Yaskawa INFORM job: DEMO_ROOF_SIDE_0625_3PAINT_37.JBI

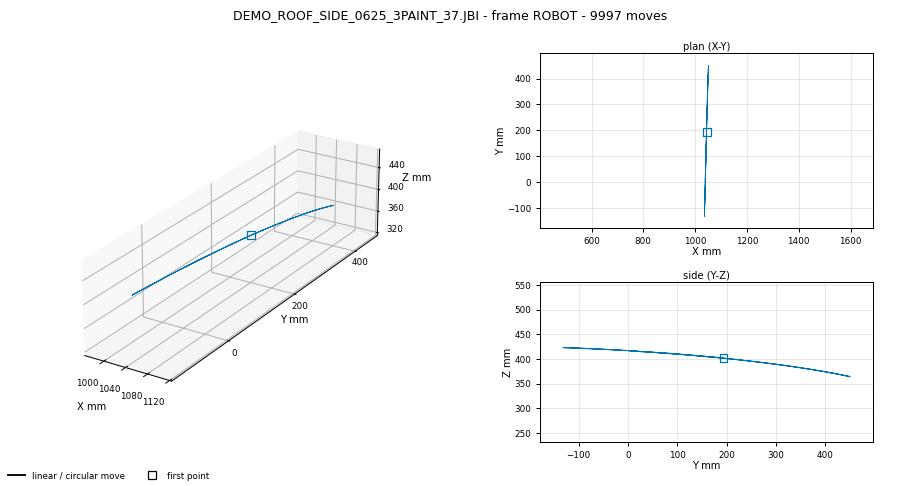
[picture p0: tool path of DEMO_ROOF_SIDE_0625_3PAINT_37.JBI in frame ROBOT, 9997 of 9997 moves have a stored position in this frame; points joined in program order, loops and branches not executed]
/JOB
//NAME DEMO_ROOF_SIDE_0625_3PAINT37
//POS
///NPOS 9997,0,0,0,0,0
///TOOL 0
///USER 0
///POSTYPE ROBOT
///RECTAN
///RCONF 1,0,0,0,0,0,0,0,0,0,0,0,0,0,0,0,0,0,0,0,0,0,0,0
C00000=1044.658,193.704,402.570,170.909,38.370,157.244
C00001=1044.653,193.455,402.594,170.907,38.368,157.244
C00002=1044.647,193.206,402.619,170.903,38.367,157.243
C00003=1044.641,192.958,402.643,170.901,38.365,157.243
C00004=1044.635,192.709,402.668,170.899,38.364,157.243
C00005=1044.628,192.460,402.692,170.895,38.362,157.242
C00006=1044.623,192.211,402.716,170.893,38.360,157.242
C00007=1044.616,191.962,402.740,170.891,38.359,157.241
C00008=1044.611,191.714,402.765,170.888,38.357,157.241
C00009=1044.604,191.465,402.789,170.885,38.355,157.241
C00010=1044.598,191.216,402.814,170.883,38.353,157.240
C00011=1044.592,190.968,402.838,170.880,38.352,157.240
C00012=1044.586,190.719,402.862,170.877,38.350,157.239
C00013=1044.580,190.470,402.886,170.875,38.348,157.239
C00014=1044.574,190.221,402.911,170.872,38.347,157.239
C00015=1044.567,189.937,402.939,170.869,38.345,157.238
C00016=1044.561,189.653,402.966,170.867,38.342,157.238
C00017=1044.553,189.368,402.994,170.863,38.341,157.237
C00018=1044.547,189.083,403.022,170.860,38.339,157.237
C00019=1044.541,188.835,403.045,170.858,38.337,157.236
C00020=1044.535,188.586,403.070,170.855,38.336,157.236
C00021=1044.529,188.337,403.094,170.853,38.334,157.236
C00022=1044.523,188.088,403.118,170.850,38.332,157.235
C00023=1044.517,187.840,403.142,170.847,38.330,157.235
C00024=1044.511,187.591,403.167,170.845,38.329,157.234
C00025=1044.505,187.343,403.191,170.843,38.327,157.234
C00026=1044.499,187.094,403.216,170.840,38.325,157.234
C00027=1044.493,186.845,403.239,170.837,38.323,157.233
C00028=1044.487,186.596,403.264,170.835,38.322,157.233
C00029=1044.481,186.347,403.287,170.832,38.320,157.232
C00030=1044.475,186.098,403.311,170.830,38.319,157.232
C00031=1044.469,185.850,403.335,170.827,38.317,157.232
C00032=1044.463,185.600,403.360,170.824,38.315,157.231
C00033=1044.457,185.352,403.383,170.822,38.313,157.231
C00034=1044.451,185.104,403.407,170.820,38.312,157.230
C00035=1044.445,184.854,403.432,170.817,38.310,157.230
C00036=1044.439,184.606,403.455,170.814,38.308,157.230
C00037=1044.433,184.357,403.480,170.812,38.307,157.229
C00038=1044.427,184.109,403.504,170.809,38.305,157.229
C00039=1044.422,183.859,403.528,170.807,38.304,157.229
C00040=1044.416,183.610,403.551,170.805,38.302,157.228
C00041=1044.409,183.361,403.575,170.801,38.300,157.228
C00042=1044.403,183.113,403.599,170.799,38.299,157.227
C00043=1044.396,182.864,403.623,170.797,38.297,157.227
C00044=1044.391,182.615,403.646,170.795,38.296,157.227
C00045=1044.384,182.366,403.670,170.791,38.294,157.226
C00046=1044.378,182.118,403.693,170.789,38.293,157.226
C00047=1044.372,181.868,403.717,170.787,38.291,157.226
C00048=1044.366,181.620,403.740,170.784,38.290,157.225
C00049=1044.358,181.371,403.764,170.781,38.289,157.225
C00050=1044.353,181.123,403.787,170.779,38.287,157.225
C00051=1044.346,180.874,403.811,170.777,38.286,157.224
C00052=1044.340,180.625,403.834,170.774,38.284,157.224
C00053=1044.334,180.376,403.857,170.771,38.283,157.224
C00054=1044.328,180.127,403.882,170.769,38.281,157.223
C00055=1044.322,179.879,403.904,170.766,38.279,157.223
C00056=1044.315,179.630,403.928,170.764,38.278,157.223
C00057=1044.309,179.381,403.951,170.762,38.276,157.222
C00058=1044.303,179.132,403.975,170.758,38.275,157.222
C00059=1044.297,178.883,403.999,170.756,38.274,157.222
C00060=1044.291,178.635,404.022,170.754,38.272,157.221
C00061=1044.284,178.386,404.045,170.752,38.271,157.221
C00062=1044.278,178.137,404.068,170.749,38.270,157.221
C00063=1044.271,177.888,404.092,170.746,38.268,157.220
C00064=1044.266,177.639,404.115,170.744,38.266,157.220
C00065=1044.260,177.391,404.139,170.741,38.265,157.219
C00066=1044.253,177.141,404.162,170.739,38.263,157.219
C00067=1044.247,176.893,404.186,170.737,38.262,157.219
C00068=1044.241,176.643,404.209,170.734,38.260,157.218
C00069=1044.235,176.394,404.232,170.731,38.259,157.218
C00070=1044.229,176.146,404.256,170.729,38.257,157.218
C00071=1044.222,175.897,404.279,170.727,38.256,157.217
C00072=1044.216,175.649,404.302,170.724,38.255,157.217
C00073=1044.210,175.400,404.325,170.722,38.253,157.217
C00074=1044.204,175.151,404.349,170.719,38.252,157.216
C00075=1044.198,174.902,404.372,170.717,38.251,157.216
C00076=1044.192,174.653,404.395,170.714,38.249,157.216
C00077=1044.186,174.405,404.419,170.712,38.248,157.215
C00078=1044.180,174.155,404.442,170.710,38.246,157.215
C00079=1044.173,173.871,404.469,170.706,38.244,157.215
C00080=1044.166,173.586,404.495,170.704,38.242,157.214
C00081=1044.158,173.301,404.521,170.701,38.241,157.214
C00082=1044.152,173.016,404.548,170.699,38.239,157.214
C00083=1044.146,172.767,404.572,170.696,38.238,157.213
C00084=1044.140,172.518,404.595,170.694,38.237,157.213
C00085=1044.133,172.270,404.618,170.692,38.235,157.212
C00086=1044.127,172.020,404.641,170.689,38.234,157.212
C00087=1044.121,171.771,404.664,170.686,38.232,157.212
C00088=1044.115,171.523,404.688,170.684,38.231,157.212
C00089=1044.109,171.274,404.710,170.682,38.229,157.211
C00090=1044.103,171.025,404.733,170.679,38.228,157.211
C00091=1044.097,170.776,404.757,170.677,38.226,157.210
C00092=1044.091,170.527,404.779,170.675,38.224,157.210
C00093=1044.085,170.279,404.803,170.672,38.223,157.210
C00094=1044.079,170.030,404.826,170.670,38.221,157.209
C00095=1044.073,169.781,404.849,170.668,38.220,157.209
C00096=1044.067,169.532,404.872,170.665,38.219,157.209
C00097=1044.061,169.283,404.895,170.662,38.217,157.208
C00098=1044.054,169.035,404.918,170.660,38.216,157.208
C00099=1044.049,168.786,404.941,170.658,38.214,157.208
C00100=1044.043,168.537,404.964,170.656,38.213,157.208
C00101=1044.037,168.287,404.987,170.653,38.212,157.207
C00102=1044.031,168.038,405.010,170.651,38.210,157.207
C00103=1044.025,167.789,405.033,170.649,38.209,157.206
C00104=1044.019,167.541,405.055,170.646,38.207,157.206
C00105=1044.013,167.293,405.079,170.644,38.206,157.206
C00106=1044.007,167.044,405.102,170.642,38.205,157.205
C00107=1044.001,166.795,405.125,170.640,38.203,157.205
C00108=1043.995,166.546,405.148,170.636,38.202,157.205
C00109=1043.989,166.296,405.171,170.634,38.200,157.204
C00110=1043.983,166.048,405.194,170.632,38.199,157.204
C00111=1043.977,165.799,405.216,170.629,38.197,157.204
C00112=1043.971,165.550,405.239,170.627,38.196,157.203
C00113=1043.965,165.301,405.262,170.625,38.194,157.203
C00114=1043.960,165.052,405.285,170.623,38.193,157.203
C00115=1043.953,164.804,405.308,170.620,38.191,157.202
C00116=1043.947,164.555,405.331,170.618,38.190,157.202
C00117=1043.942,164.306,405.354,170.616,38.188,157.202
C00118=1043.936,164.057,405.377,170.614,38.187,157.201
C00119=1043.930,163.808,405.399,170.611,38.185,157.201
C00120=1043.924,163.559,405.422,170.609,38.184,157.201
C00121=1043.917,163.310,405.445,170.607,38.182,157.200
C00122=1043.912,163.061,405.468,170.604,38.181,157.200
C00123=1043.906,162.812,405.491,170.602,38.179,157.200
C00124=1043.900,162.563,405.513,170.600,38.178,157.199
C00125=1043.894,162.315,405.536,170.598,38.177,157.199
C00126=1043.888,162.066,405.559,170.595,38.175,157.199
C00127=1043.882,161.817,405.582,170.593,38.174,157.199
C00128=1043.877,161.568,405.605,170.591,38.172,157.198
C00129=1043.870,161.319,405.627,170.589,38.171,157.198
C00130=1043.865,161.070,405.650,170.586,38.170,157.197
C00131=1043.859,160.821,405.673,170.584,38.168,157.197
C00132=1043.853,160.572,405.696,170.582,38.167,157.197
C00133=1043.847,160.323,405.718,170.580,38.165,157.197
C00134=1043.841,160.074,405.741,170.577,38.164,157.196
C00135=1043.835,159.825,405.763,170.575,38.162,157.196
C00136=1043.829,159.576,405.786,170.573,38.161,157.196
C00137=1043.823,159.328,405.808,170.571,38.160,157.195
C00138=1043.817,159.079,405.829,170.568,38.158,157.195
C00139=1043.811,158.830,405.852,170.565,38.157,157.195
C00140=1043.804,158.581,405.875,170.563,38.156,157.194
C00141=1043.799,158.332,405.898,170.561,38.155,157.194
C00142=1043.792,158.083,405.919,170.558,38.153,157.194
C00143=1043.785,157.798,405.945,170.556,38.152,157.193
C00144=1043.778,157.513,405.970,170.554,38.150,157.193
C00145=1043.771,157.228,405.996,170.550,38.149,157.193
C00146=1043.764,156.941,406.022,170.548,38.147,157.192
C00147=1043.758,156.693,406.045,170.546,38.146,157.192
C00148=1043.752,156.444,406.066,170.544,38.145,157.192
C00149=1043.746,156.195,406.089,170.541,38.143,157.191
C00150=1043.740,155.946,406.111,170.539,38.142,157.191
C00151=1043.733,155.697,406.133,170.537,38.141,157.191
C00152=1043.728,155.448,406.156,170.535,38.140,157.191
C00153=1043.722,155.199,406.178,170.532,38.138,157.190
C00154=1043.715,154.950,406.200,170.530,38.137,157.190
C00155=1043.710,154.701,406.222,170.528,38.136,157.190
C00156=1043.703,154.452,406.245,170.526,38.135,157.189
C00157=1043.698,154.204,406.266,170.523,38.133,157.189
C00158=1043.692,153.955,406.289,170.521,38.132,157.189
C00159=1043.686,153.706,406.311,170.519,38.130,157.189
C00160=1043.679,153.457,406.333,170.517,38.129,157.188
C00161=1043.673,153.208,406.355,170.515,38.128,157.188
C00162=1043.667,152.959,406.378,170.512,38.126,157.188
C00163=1043.661,152.710,406.399,170.510,38.125,157.187
C00164=1043.655,152.461,406.422,170.508,38.124,157.187
C00165=1043.649,152.212,406.443,170.506,38.123,157.187
C00166=1043.642,151.963,406.466,170.503,38.122,157.187
C00167=1043.637,151.714,406.488,170.501,38.121,157.186
C00168=1043.631,151.465,406.509,170.499,38.119,157.186
C00169=1043.624,151.216,406.532,170.497,38.118,157.186
C00170=1043.618,150.967,406.553,170.494,38.116,157.185
C00171=1043.611,150.718,406.576,170.492,38.115,157.185
C00172=1043.607,150.469,406.598,170.490,38.114,157.185
C00173=1043.600,150.220,406.619,170.488,38.112,157.184
C00174=1043.594,149.972,406.642,170.485,38.111,157.184
C00175=1043.588,149.722,406.663,170.483,38.110,157.184
C00176=1043.582,149.473,406.685,170.481,38.109,157.184
C00177=1043.576,149.224,406.708,170.479,38.108,157.183
C00178=1043.570,148.975,406.729,170.478,38.107,157.183
C00179=1043.564,148.726,406.751,170.475,38.105,157.183
C00180=1043.558,148.478,406.773,170.473,38.104,157.182
C00181=1043.552,148.229,406.795,170.471,38.102,157.182
C00182=1043.545,147.980,406.816,170.469,38.101,157.182
C00183=1043.539,147.731,406.839,170.466,38.100,157.182
C00184=1043.533,147.482,406.860,170.464,38.099,157.181
C00185=1043.527,147.232,406.883,170.462,38.098,157.181
C00186=1043.521,146.983,406.904,170.460,38.097,157.181
C00187=1043.515,146.734,406.926,170.457,38.095,157.180
C00188=1043.509,146.486,406.948,170.455,38.094,157.180
C00189=1043.503,146.237,406.969,170.453,38.092,157.180
C00190=1043.496,145.988,406.990,170.451,38.091,157.180
C00191=1043.490,145.739,407.012,170.448,38.090,157.179
C00192=1043.484,145.489,407.034,170.446,38.089,157.179
C00193=1043.478,145.240,407.055,170.444,38.088,157.179
C00194=1043.472,144.992,407.077,170.442,38.087,157.178
C00195=1043.466,144.743,407.099,170.440,38.086,157.178
C00196=1043.459,144.494,407.121,170.437,38.084,157.178
C00197=1043.453,144.245,407.142,170.435,38.083,157.178
C00198=1043.447,143.996,407.164,170.433,38.082,157.177
C00199=1043.441,143.746,407.186,170.432,38.081,157.177
C00200=1043.435,143.498,407.207,170.430,38.080,157.177
C00201=1043.429,143.249,407.228,170.427,38.078,157.177
C00202=1043.423,142.999,407.250,170.425,38.077,157.176
C00203=1043.417,142.751,407.272,170.423,38.076,157.176
C00204=1043.410,142.502,407.294,170.421,38.074,157.176
C00205=1043.405,142.253,407.315,170.418,38.073,157.175
C00206=1043.399,142.004,407.337,170.416,38.072,157.175
C00207=1043.391,141.718,407.361,170.414,38.071,157.175
C00208=1043.385,141.433,407.386,170.412,38.070,157.175
C00209=1043.378,141.146,407.411,170.408,38.068,157.174
C00210=1043.370,140.862,407.435,170.406,38.067,157.174
C00211=1043.364,140.612,407.457,170.404,38.066,157.174
C00212=1043.358,140.363,407.478,170.402,38.064,157.173
C00213=1043.352,140.115,407.499,170.401,38.063,157.173
C00214=1043.346,139.865,407.521,170.398,38.062,157.173
C00215=1043.340,139.616,407.543,170.396,38.060,157.173
C00216=1043.334,139.367,407.564,170.394,38.059,157.172
C00217=1043.328,139.119,407.586,170.392,38.058,157.172
C00218=1043.321,138.870,407.607,170.389,38.057,157.172
C00219=1043.315,138.620,407.628,170.387,38.056,157.171
C00220=1043.309,138.371,407.649,170.385,38.054,157.171
C00221=1043.304,138.122,407.671,170.383,38.053,157.171
C00222=1043.298,137.873,407.692,170.381,38.052,157.171
C00223=1043.291,137.624,407.713,170.378,38.051,157.170
C00224=1043.285,137.376,407.734,170.377,38.050,157.170
C00225=1043.279,137.126,407.756,170.375,38.049,157.170
C00226=1043.273,136.877,407.778,170.373,38.047,157.170
C00227=1043.266,136.628,407.798,170.371,38.047,157.169
C00228=1043.261,136.379,407.819,170.368,38.046,157.169
C00229=1043.255,136.130,407.841,170.366,38.045,157.169
C00230=1043.248,135.881,407.862,170.364,38.043,157.169
C00231=1043.242,135.632,407.883,170.362,38.042,157.168
C00232=1043.236,135.383,407.904,170.359,38.041,157.168
C00233=1043.229,135.134,407.925,170.357,38.040,157.168
C00234=1043.224,134.885,407.947,170.356,38.039,157.168
C00235=1043.218,134.636,407.968,170.354,38.037,157.167
C00236=1043.211,134.387,407.988,170.352,38.036,157.167
C00237=1043.206,134.138,408.010,170.349,38.035,157.167
C00238=1043.199,133.889,408.031,170.347,38.034,157.167
C00239=1043.192,133.640,408.052,170.345,38.033,157.166
C00240=1043.187,133.391,408.073,170.343,38.032,157.166
C00241=1043.181,133.142,408.095,170.341,38.030,157.166
C00242=1043.174,132.893,408.116,170.338,38.029,157.165
C00243=1043.169,132.644,408.136,170.337,38.028,157.165
C00244=1043.163,132.394,408.158,170.335,38.027,157.165
C00245=1043.156,132.146,408.179,170.333,38.026,157.165
C00246=1043.151,131.896,408.199,170.330,38.025,157.164
C00247=1043.144,131.647,408.221,170.328,38.023,157.164
C00248=1043.138,131.399,408.242,170.326,38.022,157.164
C00249=1043.132,131.149,408.263,170.324,38.021,157.164
C00250=1043.125,130.900,408.284,170.323,38.020,157.163
C00251=1043.120,130.651,408.304,170.321,38.019,157.163
C00252=1043.113,130.402,408.325,170.318,38.018,157.163
C00253=1043.107,130.152,408.346,170.316,38.017,157.163
C00254=1043.101,129.904,408.367,170.314,38.016,157.162
C00255=1043.094,129.655,408.387,170.312,38.015,157.162
C00256=1043.088,129.405,408.409,170.309,38.013,157.162
C00257=1043.082,129.157,408.429,170.307,38.013,157.162
C00258=1043.075,128.908,408.450,170.305,38.012,157.161
C00259=1043.070,128.659,408.470,170.304,38.011,157.161
C00260=1043.063,128.410,408.491,170.302,38.009,157.161
C00261=1043.057,128.160,408.512,170.300,38.008,157.161
C00262=1043.051,127.912,408.533,170.297,38.008,157.161
C00263=1043.044,127.662,408.553,170.295,38.006,157.160
C00264=1043.039,127.414,408.575,170.293,38.005,157.160
C00265=1043.032,127.164,408.595,170.291,38.004,157.160
C00266=1043.025,126.915,408.616,170.289,38.003,157.159
C00267=1043.020,126.666,408.637,170.287,38.002,157.159
C00268=1043.013,126.417,408.658,170.285,38.001,157.159
C00269=1043.007,126.168,408.678,170.283,38.000,157.159
C00270=1043.001,125.919,408.698,170.281,37.999,157.159
C00271=1042.994,125.633,408.722,170.279,37.998,157.158
C00272=1042.987,125.347,408.746,170.276,37.996,157.158
C00273=1042.980,125.062,408.770,170.274,37.995,157.158
C00274=1042.972,124.775,408.793,170.271,37.994,157.157
C00275=1042.966,124.527,408.814,170.270,37.993,157.157
C00276=1042.960,124.277,408.835,170.268,37.992,157.157
C00277=1042.954,124.028,408.855,170.265,37.991,157.157
C00278=1042.947,123.779,408.876,170.263,37.989,157.156
C00279=1042.942,123.530,408.896,170.261,37.988,157.156
C00280=1042.936,123.281,408.917,170.259,37.987,157.156
C00281=1042.929,123.032,408.937,170.257,37.987,157.156
C00282=1042.923,122.783,408.958,170.255,37.985,157.156
C00283=1042.917,122.534,408.978,170.253,37.984,157.155
C00284=1042.911,122.285,408.999,170.251,37.983,157.155
C00285=1042.905,122.036,409.020,170.249,37.982,157.155
C00286=1042.899,121.786,409.040,170.247,37.981,157.154
C00287=1042.893,121.538,409.060,170.244,37.979,157.154
C00288=1042.886,121.289,409.081,170.243,37.979,157.154
C00289=1042.881,121.039,409.102,170.241,37.978,157.154
C00290=1042.874,120.790,409.122,170.239,37.977,157.154
C00291=1042.868,120.541,409.142,170.237,37.975,157.153
C00292=1042.862,120.293,409.163,170.234,37.974,157.153
C00293=1042.856,120.043,409.184,170.233,37.973,157.153
C00294=1042.850,119.794,409.203,170.231,37.972,157.152
C00295=1042.844,119.544,409.224,170.229,37.971,157.152
C00296=1042.838,119.296,409.244,170.227,37.970,157.152
C00297=1042.831,119.047,409.265,170.224,37.969,157.152
C00298=1042.825,118.798,409.285,170.222,37.968,157.152
C00299=1042.820,118.549,409.306,170.221,37.966,157.151
C00300=1042.813,118.299,409.326,170.219,37.965,157.151
C00301=1042.807,118.051,409.346,170.217,37.964,157.151
C00302=1042.801,117.801,409.367,170.214,37.963,157.150
C00303=1042.795,117.553,409.388,170.212,37.962,157.150
C00304=1042.788,117.303,409.408,170.211,37.961,157.150
C00305=1042.782,117.054,409.428,170.209,37.960,157.150
C00306=1042.777,116.805,409.449,170.207,37.959,157.150
C00307=1042.771,116.556,409.469,170.204,37.958,157.149
C00308=1042.765,116.307,409.489,170.202,37.956,157.149
C00309=1042.759,116.058,409.509,170.201,37.955,157.149
C00310=1042.753,115.808,409.530,170.199,37.954,157.149
C00311=1042.747,115.559,409.550,170.197,37.953,157.148
C00312=1042.740,115.311,409.570,170.195,37.952,157.148
C00313=1042.735,115.061,409.591,170.192,37.951,157.148
C00314=1042.729,114.812,409.611,170.191,37.950,157.148
C00315=1042.723,114.564,409.631,170.189,37.949,157.147
C00316=1042.716,114.314,409.652,170.187,37.948,157.147
C00317=1042.711,114.065,409.672,170.184,37.946,157.147
C00318=1042.705,113.816,409.692,170.183,37.945,157.147
C00319=1042.698,113.567,409.712,170.181,37.944,157.146
C00320=1042.692,113.318,409.732,170.179,37.943,157.146
C00321=1042.686,113.068,409.753,170.177,37.942,157.146
C00322=1042.680,112.820,409.773,170.175,37.941,157.146
C00323=1042.674,112.571,409.793,170.173,37.940,157.145
C00324=1042.667,112.321,409.812,170.171,37.939,157.145
C00325=1042.661,112.072,409.832,170.169,37.938,157.145
C00326=1042.655,111.823,409.852,170.167,37.937,157.145
C00327=1042.649,111.573,409.872,170.165,37.936,157.144
C00328=1042.643,111.325,409.892,170.163,37.935,157.144
C00329=1042.637,111.076,409.912,170.161,37.934,157.144
C00330=1042.630,110.826,409.933,170.159,37.933,157.144
C00331=1042.624,110.577,409.953,170.157,37.932,157.144
C00332=1042.618,110.329,409.973,170.155,37.930,157.143
C00333=1042.612,110.079,409.992,170.154,37.930,157.143
C00334=1042.606,109.830,410.012,170.151,37.929,157.143
C00335=1042.599,109.544,410.035,170.149,37.928,157.143
C00336=1042.591,109.257,410.058,170.147,37.926,157.142
C00337=1042.584,108.971,410.081,170.144,37.925,157.142
C00338=1042.577,108.686,410.103,170.142,37.924,157.142
C00339=1042.571,108.437,410.123,170.140,37.923,157.142
C00340=1042.564,108.187,410.143,170.138,37.922,157.141
C00341=1042.558,107.938,410.163,170.136,37.921,157.141
C00342=1042.553,107.689,410.183,170.134,37.920,157.141
C00343=1042.546,107.441,410.202,170.132,37.919,157.141
C00344=1042.539,107.191,410.222,170.130,37.918,157.140
C00345=1042.533,106.942,410.242,170.128,37.917,157.140
C00346=1042.528,106.693,410.261,170.126,37.916,157.140
C00347=1042.521,106.443,410.282,170.124,37.915,157.140
C00348=1042.515,106.194,410.302,170.122,37.914,157.140
C00349=1042.509,105.945,410.320,170.121,37.913,157.139
C00350=1042.503,105.696,410.340,170.118,37.912,157.139
C00351=1042.496,105.447,410.361,170.116,37.911,157.139
C00352=1042.490,105.198,410.380,170.114,37.910,157.139
C00353=1042.484,104.949,410.400,170.113,37.909,157.139
C00354=1042.478,104.700,410.420,170.111,37.908,157.138
C00355=1042.471,104.450,410.439,170.109,37.907,157.138
C00356=1042.465,104.201,410.459,170.106,37.906,157.138
C00357=1042.459,103.952,410.479,170.104,37.905,157.138
C00358=1042.454,103.703,410.498,170.103,37.904,157.137
C00359=1042.447,103.454,410.518,170.101,37.903,157.137
C00360=1042.441,103.204,410.537,170.099,37.902,157.137
C00361=1042.435,102.956,410.557,170.096,37.901,157.137
C00362=1042.429,102.707,410.577,170.095,37.900,157.136
C00363=1042.423,102.457,410.596,170.093,37.899,157.136
C00364=1042.416,102.208,410.617,170.091,37.897,157.136
C00365=1042.411,101.958,410.636,170.089,37.897,157.136
C00366=1042.404,101.710,410.655,170.087,37.896,157.135
C00367=1042.398,101.461,410.675,170.085,37.894,157.135
C00368=1042.392,101.212,410.694,170.083,37.893,157.135
C00369=1042.386,100.962,410.715,170.081,37.893,157.135
C00370=1042.380,100.713,410.734,170.079,37.892,157.135
C00371=1042.373,100.464,410.753,170.078,37.890,157.134
C00372=1042.368,100.215,410.773,170.076,37.890,157.134
C00373=1042.362,99.966,410.792,170.073,37.889,157.134
C00374=1042.355,99.716,410.811,170.071,37.887,157.134
C00375=1042.349,99.467,410.831,170.070,37.887,157.134
C00376=1042.342,99.218,410.850,170.068,37.886,157.133
C00377=1042.337,98.969,410.869,170.066,37.884,157.133
C00378=1042.330,98.720,410.889,170.063,37.884,157.133
C00379=1042.323,98.470,410.908,170.061,37.883,157.133
C00380=1042.317,98.222,410.928,170.060,37.882,157.132
C00381=1042.311,97.972,410.947,170.058,37.881,157.132
C00382=1042.305,97.723,410.966,170.056,37.880,157.132
C00383=1042.299,97.474,410.986,170.054,37.879,157.132
C00384=1042.292,97.224,411.005,170.051,37.878,157.132
C00385=1042.286,96.976,411.024,170.050,37.877,157.131
C00386=1042.280,96.726,411.044,170.048,37.876,157.131
C00387=1042.274,96.477,411.062,170.046,37.875,157.131
C00388=1042.268,96.228,411.082,170.044,37.874,157.131
C00389=1042.261,95.979,411.101,170.043,37.873,157.130
C00390=1042.255,95.730,411.120,170.040,37.872,157.130
C00391=1042.248,95.480,411.140,170.038,37.871,157.130
C00392=1042.242,95.231,411.159,170.036,37.870,157.130
C00393=1042.236,94.982,411.178,170.035,37.869,157.130
C00394=1042.230,94.732,411.197,170.033,37.868,157.129
C00395=1042.224,94.484,411.216,170.031,37.867,157.129
C00396=1042.218,94.235,411.236,170.028,37.866,157.129
C00397=1042.212,93.985,411.255,170.026,37.866,157.129
C00398=1042.205,93.737,411.274,170.025,37.864,157.129
C00399=1042.198,93.450,411.296,170.023,37.863,157.128
C00400=1042.191,93.165,411.318,170.021,37.862,157.128
C00401=1042.184,92.878,411.340,170.018,37.861,157.128
C00402=1042.177,92.592,411.362,170.016,37.860,157.127
C00403=1042.171,92.343,411.382,170.014,37.859,157.127
C00404=1042.165,92.094,411.401,170.012,37.858,157.127
C00405=1042.158,91.845,411.419,170.010,37.857,157.127
C00406=1042.153,91.595,411.439,170.009,37.856,157.127
C00407=1042.146,91.346,411.457,170.006,37.855,157.126
C00408=1042.140,91.097,411.477,170.004,37.854,157.126
C00409=1042.134,90.848,411.496,170.002,37.853,157.126
C00410=1042.128,90.599,411.515,170.001,37.852,157.126
C00411=1042.122,90.350,411.534,169.999,37.851,157.126
C00412=1042.116,90.100,411.553,169.997,37.850,157.125
C00413=1042.109,89.850,411.572,169.994,37.849,157.125
C00414=1042.103,89.601,411.591,169.993,37.848,157.125
C00415=1042.096,89.353,411.610,169.991,37.847,157.125
C00416=1042.090,89.103,411.629,169.989,37.846,157.124
C00417=1042.084,88.854,411.648,169.987,37.845,157.124
C00418=1042.077,88.605,411.667,169.985,37.844,157.124
C00419=1042.071,88.356,411.685,169.984,37.844,157.124
C00420=1042.065,88.106,411.704,169.981,37.842,157.124
C00421=1042.059,87.857,411.723,169.979,37.842,157.124
C00422=1042.052,87.608,411.742,169.977,37.841,157.123
C00423=1042.046,87.359,411.760,169.976,37.840,157.123
C00424=1042.040,87.110,411.780,169.974,37.839,157.123
C00425=1042.034,86.861,411.798,169.972,37.838,157.123
C00426=1042.027,86.611,411.817,169.969,37.837,157.122
C00427=1042.021,86.362,411.836,169.967,37.836,157.122
C00428=1042.015,86.113,411.854,169.966,37.835,157.122
C00429=1042.009,85.864,411.874,169.964,37.834,157.122
C00430=1042.003,85.615,411.892,169.962,37.834,157.122
C00431=1041.996,85.365,411.911,169.960,37.832,157.121
C00432=1041.990,85.116,411.929,169.958,37.832,157.121
C00433=1041.984,84.867,411.949,169.956,37.831,157.121
C00434=1041.978,84.618,411.967,169.954,37.829,157.121
C00435=1041.971,84.369,411.986,169.952,37.829,157.121
C00436=1041.965,84.120,412.005,169.951,37.828,157.120
C00437=1041.958,83.870,412.023,169.949,37.827,157.120
C00438=1041.953,83.620,412.042,169.946,37.826,157.120
C00439=1041.946,83.371,412.060,169.944,37.825,157.120
C00440=1041.940,83.122,412.079,169.943,37.824,157.120
C00441=1041.934,82.873,412.098,169.941,37.823,157.119
C00442=1041.927,82.624,412.116,169.939,37.822,157.119
C00443=1041.922,82.374,412.136,169.937,37.821,157.119
C00444=1041.915,82.125,412.154,169.936,37.820,157.119
C00445=1041.909,81.876,412.173,169.933,37.819,157.119
C00446=1041.902,81.627,412.192,169.931,37.818,157.118
C00447=1041.896,81.377,412.210,169.929,37.818,157.118
C00448=1041.890,81.128,412.229,169.928,37.816,157.118
C00449=1041.884,80.879,412.247,169.926,37.816,157.118
C00450=1041.878,80.630,412.266,169.924,37.815,157.118
C00451=1041.872,80.381,412.284,169.921,37.813,157.117
C00452=1041.866,80.132,412.302,169.920,37.813,157.117
C00453=1041.860,79.882,412.322,169.918,37.812,157.117
C00454=1041.854,79.633,412.340,169.916,37.811,157.117
C00455=1041.847,79.384,412.359,169.914,37.810,157.116
C00456=1041.841,79.135,412.377,169.913,37.809,157.116
C00457=1041.835,78.885,412.395,169.910,37.808,157.116
C00458=1041.828,78.636,412.414,169.908,37.807,157.116
C00459=1041.822,78.386,412.433,169.906,37.806,157.116
C00460=1041.816,78.137,412.452,169.905,37.805,157.115
C00461=1041.810,77.888,412.470,169.903,37.804,157.115
C00462=1041.804,77.639,412.488,169.901,37.803,157.115
C00463=1041.796,77.353,412.509,169.898,37.802,157.115
C00464=1041.789,77.067,412.531,169.896,37.801,157.115
C00465=1041.782,76.781,412.551,169.894,37.800,157.114
C00466=1041.775,76.495,412.572,169.892,37.799,157.114
C00467=1041.769,76.245,412.591,169.890,37.798,157.114
C00468=1041.762,75.996,412.610,169.888,37.797,157.114
C00469=1041.756,75.747,412.628,169.886,37.796,157.113
C00470=1041.750,75.498,412.646,169.884,37.796,157.113
C00471=1041.744,75.248,412.664,169.882,37.794,157.113
C00472=1041.738,74.999,412.683,169.880,37.794,157.113
C00473=1041.730,74.750,412.701,169.879,37.793,157.113
C00474=1041.724,74.501,412.719,169.877,37.792,157.113
C00475=1041.718,74.252,412.737,169.875,37.791,157.112
C00476=1041.712,74.002,412.755,169.872,37.790,157.112
C00477=1041.706,73.753,412.773,169.871,37.789,157.112
C00478=1041.700,73.504,412.792,169.869,37.788,157.112
C00479=1041.693,73.255,412.810,169.867,37.787,157.112
C00480=1041.687,73.005,412.829,169.865,37.787,157.111
C00481=1041.681,72.756,412.847,169.863,37.785,157.111
C00482=1041.674,72.507,412.865,169.861,37.785,157.111
C00483=1041.669,72.258,412.883,169.859,37.784,157.111
C00484=1041.662,72.008,412.901,169.857,37.783,157.111
C00485=1041.656,71.759,412.919,169.855,37.782,157.110
C00486=1041.649,71.510,412.937,169.854,37.781,157.110
C00487=1041.643,71.260,412.955,169.852,37.780,157.110
C00488=1041.637,71.011,412.974,169.850,37.779,157.110
C00489=1041.631,70.762,412.992,169.847,37.778,157.110
C00490=1041.625,70.513,413.010,169.846,37.778,157.109
C00491=1041.619,70.263,413.028,169.844,37.776,157.109
C00492=1041.612,70.014,413.047,169.842,37.775,157.109
C00493=1041.606,69.765,413.064,169.840,37.775,157.109
C00494=1041.600,69.515,413.082,169.839,37.773,157.109
C00495=1041.593,69.266,413.100,169.836,37.773,157.108
C00496=1041.587,69.017,413.118,169.834,37.772,157.108
C00497=1041.581,68.768,413.137,169.832,37.771,157.108
C00498=1041.575,68.519,413.154,169.831,37.771,157.108
C00499=1041.568,68.269,413.172,169.829,37.769,157.108
C00500=1041.562,68.020,413.190,169.827,37.769,157.107
C00501=1041.556,67.770,413.208,169.825,37.768,157.107
C00502=1041.549,67.522,413.226,169.822,37.767,157.107
C00503=1041.543,67.272,413.244,169.821,37.766,157.107
C00504=1041.537,67.023,413.262,169.819,37.765,157.107
C00505=1041.531,66.773,413.281,169.817,37.764,157.106
C00506=1041.524,66.524,413.298,169.815,37.763,157.106
C00507=1041.518,66.275,413.315,169.814,37.762,157.106
C00508=1041.512,66.025,413.333,169.812,37.762,157.106
C00509=1041.505,65.776,413.351,169.809,37.760,157.106
C00510=1041.499,65.527,413.369,169.807,37.760,157.106
C00511=1041.493,65.278,413.387,169.805,37.759,157.105
C00512=1041.486,65.029,413.405,169.804,37.758,157.105
C00513=1041.480,64.779,413.423,169.802,37.757,157.105
C00514=1041.475,64.530,413.441,169.800,37.756,157.105
C00515=1041.468,64.281,413.458,169.798,37.756,157.105
C00516=1041.461,64.032,413.477,169.796,37.754,157.104
C00517=1041.455,63.782,413.494,169.794,37.754,157.104
C00518=1041.449,63.533,413.511,169.792,37.753,157.104
C00519=1041.443,63.283,413.529,169.790,37.752,157.104
C00520=1041.436,63.034,413.547,169.788,37.752,157.104
C00521=1041.429,62.784,413.564,169.787,37.750,157.103
C00522=1041.423,62.536,413.582,169.785,37.750,157.103
C00523=1041.416,62.287,413.600,169.782,37.749,157.103
C00524=1041.410,62.037,413.618,169.780,37.748,157.103
C00525=1041.403,61.787,413.635,169.778,37.747,157.103
C00526=1041.397,61.539,413.652,169.777,37.747,157.103
C00527=1041.390,61.252,413.672,169.775,37.746,157.102
C00528=1041.382,60.965,413.693,169.772,37.745,157.102
C00529=1041.375,60.679,413.712,169.770,37.744,157.102
C00530=1041.367,60.393,413.733,169.767,37.743,157.102
C00531=1041.362,60.144,413.750,169.766,37.742,157.102
C00532=1041.355,59.894,413.768,169.764,37.742,157.101
C00533=1041.348,59.646,413.786,169.762,37.741,157.101
C00534=1041.342,59.397,413.803,169.760,37.740,157.101
C00535=1041.336,59.147,413.821,169.758,37.739,157.101
C00536=1041.329,58.897,413.839,169.757,37.739,157.101
C00537=1041.323,58.649,413.856,169.754,37.737,157.101
C00538=1041.316,58.399,413.873,169.752,37.737,157.100
C00539=1041.310,58.149,413.891,169.750,37.736,157.100
C00540=1041.304,57.901,413.908,169.748,37.735,157.100
C00541=1041.298,57.651,413.926,169.747,37.734,157.100
C00542=1041.291,57.402,413.943,169.745,37.733,157.100
C00543=1041.285,57.153,413.960,169.743,37.733,157.100
C00544=1041.279,56.903,413.978,169.741,37.732,157.099
C00545=1041.272,56.654,413.995,169.738,37.731,157.099
C00546=1041.265,56.405,414.012,169.737,37.730,157.099
C00547=1041.259,56.155,414.030,169.735,37.730,157.099
C00548=1041.253,55.906,414.048,169.733,37.728,157.099
C00549=1041.247,55.656,414.064,169.731,37.728,157.098
C00550=1041.240,55.407,414.082,169.729,37.727,157.098
C00551=1041.234,55.158,414.099,169.728,37.726,157.098
C00552=1041.228,54.908,414.117,169.725,37.726,157.098
C00553=1041.221,54.659,414.134,169.723,37.724,157.098
C00554=1041.215,54.410,414.151,169.721,37.724,157.098
C00555=1041.209,54.160,414.169,169.719,37.723,157.097
C00556=1041.203,53.912,414.186,169.718,37.722,157.097
C00557=1041.196,53.662,414.204,169.716,37.721,157.097
C00558=1041.190,53.413,414.221,169.714,37.720,157.097
C00559=1041.183,53.164,414.238,169.711,37.720,157.097
C00560=1041.178,52.913,414.255,169.709,37.719,157.096
C00561=1041.171,52.665,414.272,169.708,37.718,157.096
C00562=1041.164,52.415,414.290,169.706,37.717,157.096
C00563=1041.159,52.166,414.307,169.704,37.717,157.096
C00564=1041.152,51.917,414.325,169.702,37.715,157.096
C00565=1041.146,51.668,414.342,169.701,37.715,157.096
C00566=1041.140,51.418,414.359,169.698,37.714,157.095
C00567=1041.134,51.169,414.376,169.696,37.713,157.095
C00568=1041.127,50.919,414.393,169.694,37.712,157.095
C00569=1041.121,50.670,414.411,169.692,37.711,157.095
C00570=1041.114,50.421,414.428,169.691,37.711,157.095
C00571=1041.108,50.171,414.445,169.689,37.709,157.094
C00572=1041.102,49.922,414.462,169.687,37.709,157.094
C00573=1041.096,49.672,414.479,169.685,37.708,157.094
C00574=1041.089,49.424,414.496,169.682,37.707,157.094
C00575=1041.083,49.174,414.514,169.681,37.706,157.094
C00576=1041.077,48.925,414.531,169.679,37.705,157.094
C00577=1041.071,48.676,414.548,169.677,37.705,157.093
C00578=1041.065,48.426,414.566,169.675,37.703,157.093
C00579=1041.059,48.177,414.582,169.673,37.703,157.093
C00580=1041.052,47.927,414.599,169.672,37.702,157.093
C00581=1041.047,47.678,414.617,169.669,37.701,157.093
C00582=1041.040,47.429,414.634,169.667,37.701,157.092
C00583=1041.034,47.180,414.650,169.665,37.699,157.092
C00584=1041.028,46.930,414.668,169.664,37.699,157.092
C00585=1041.021,46.681,414.685,169.662,37.697,157.092
C00586=1041.015,46.431,414.702,169.660,37.697,157.092
C00587=1041.009,46.182,414.719,169.658,37.696,157.091
C00588=1041.003,45.933,414.736,169.655,37.695,157.091
C00589=1040.996,45.683,414.753,169.654,37.695,157.091
C00590=1040.991,45.434,414.771,169.652,37.693,157.091
C00591=1040.985,45.188,414.788,169.650,37.693,157.091
C00592=1040.979,44.943,414.804,169.648,37.692,157.091
C00593=1040.972,44.698,414.821,169.647,37.691,157.090
C00594=1040.967,44.452,414.837,169.645,37.690,157.090
C00595=1040.960,44.206,414.854,169.642,37.689,157.090
C00596=1040.955,43.961,414.871,169.640,37.689,157.090
C00597=1040.948,43.716,414.888,169.639,37.687,157.090
C00598=1040.942,43.471,414.904,169.637,37.687,157.089
C00599=1040.936,43.221,414.921,169.635,37.686,157.089
C00600=1040.929,42.972,414.939,169.633,37.685,157.089
C00601=1040.924,42.722,414.955,169.631,37.684,157.089
C00602=1040.917,42.473,414.972,169.629,37.683,157.089
C00603=1040.911,42.224,414.988,169.627,37.683,157.089
C00604=1040.904,41.974,415.006,169.625,37.682,157.088
C00605=1040.898,41.725,415.022,169.623,37.681,157.088
C00606=1040.892,41.476,415.039,169.621,37.680,157.088
C00607=1040.885,41.226,415.056,169.619,37.680,157.088
C00608=1040.879,40.977,415.073,169.618,37.678,157.088
C00609=1040.872,40.727,415.089,169.616,37.678,157.088
C00610=1040.866,40.479,415.106,169.613,37.677,157.087
C00611=1040.860,40.229,415.122,169.611,37.676,157.087
C00612=1040.854,39.979,415.139,169.609,37.675,157.087
C00613=1040.847,39.730,415.156,169.607,37.675,157.087
C00614=1040.841,39.481,415.172,169.606,37.674,157.087
C00615=1040.835,39.231,415.190,169.604,37.673,157.087
C00616=1040.829,38.982,415.206,169.602,37.672,157.086
C00617=1040.822,38.733,415.224,169.600,37.671,157.086
C00618=1040.816,38.483,415.240,169.597,37.671,157.086
C00619=1040.811,38.234,415.256,169.596,37.670,157.086
C00620=1040.804,37.984,415.274,169.594,37.669,157.086
C00621=1040.798,37.735,415.290,169.592,37.668,157.085
C00622=1040.792,37.486,415.306,169.590,37.668,157.085
C00623=1040.785,37.236,415.324,169.588,37.666,157.085
C00624=1040.778,36.987,415.339,169.586,37.666,157.085
C00625=1040.772,36.738,415.355,169.585,37.665,157.085
C00626=1040.765,36.489,415.373,169.582,37.665,157.085
C00627=1040.759,36.239,415.389,169.580,37.664,157.085
C00628=1040.753,35.990,415.405,169.578,37.663,157.084
C00629=1040.747,35.740,415.422,169.576,37.662,157.084
C00630=1040.740,35.491,415.438,169.574,37.662,157.084
C00631=1040.734,35.242,415.455,169.572,37.661,157.084
C00632=1040.727,34.992,415.471,169.571,37.660,157.084
C00633=1040.721,34.743,415.487,169.569,37.659,157.084
C00634=1040.715,34.494,415.504,169.566,37.659,157.083
C00635=1040.707,34.199,415.524,169.564,37.658,157.083
C00636=1040.700,33.904,415.543,169.561,37.657,157.083
C00637=1040.693,33.610,415.563,169.559,37.656,157.083
C00638=1040.685,33.315,415.582,169.557,37.655,157.083
C00639=1040.679,33.066,415.597,169.555,37.655,157.082
C00640=1040.672,32.817,415.615,169.553,37.654,157.082
C00641=1040.666,32.568,415.631,169.551,37.653,157.082
C00642=1040.660,32.318,415.647,169.549,37.652,157.082
C00643=1040.653,32.068,415.664,169.547,37.652,157.082
C00644=1040.647,31.819,415.679,169.545,37.651,157.082
C00645=1040.641,31.570,415.696,169.543,37.650,157.081
C00646=1040.635,31.320,415.712,169.541,37.649,157.081
C00647=1040.628,31.071,415.729,169.539,37.649,157.081
C00648=1040.621,30.822,415.745,169.538,37.648,157.081
C00649=1040.615,30.573,415.761,169.535,37.647,157.081
C00650=1040.609,30.323,415.778,169.533,37.646,157.081
C00651=1040.603,30.073,415.794,169.531,37.646,157.081
C00652=1040.597,29.824,415.810,169.529,37.645,157.080
C00653=1040.590,29.575,415.826,169.527,37.644,157.080
C00654=1040.584,29.326,415.842,169.525,37.643,157.080
C00655=1040.576,29.039,415.861,169.523,37.643,157.080
C00656=1040.570,28.752,415.881,169.521,37.642,157.080
C00657=1040.562,28.465,415.898,169.518,37.641,157.079
C00658=1040.555,28.179,415.917,169.516,37.640,157.079
C00659=1040.549,27.930,415.933,169.514,37.639,157.079
C00660=1040.542,27.680,415.949,169.512,37.639,157.079
C00661=1040.536,27.430,415.966,169.510,37.638,157.079
C00662=1040.530,27.181,415.982,169.508,37.637,157.079
C00663=1040.523,26.932,415.998,169.506,37.636,157.078
C00664=1040.517,26.683,416.014,169.505,37.636,157.078
C00665=1040.511,26.433,416.030,169.503,37.635,157.078
C00666=1040.504,26.184,416.046,169.500,37.634,157.078
C00667=1040.498,25.934,416.062,169.498,37.634,157.078
C00668=1040.491,25.685,416.078,169.496,37.633,157.078
C00669=1040.485,25.435,416.094,169.494,37.632,157.078
C00670=1040.478,25.186,416.110,169.492,37.632,157.077
C00671=1040.473,24.936,416.126,169.490,37.631,157.077
C00672=1040.467,24.687,416.142,169.488,37.630,157.077
C00673=1040.460,24.438,416.158,169.487,37.630,157.077
C00674=1040.454,24.188,416.174,169.485,37.629,157.077
C00675=1040.447,23.939,416.190,169.482,37.628,157.077
C00676=1040.441,23.689,416.206,169.480,37.627,157.076
C00677=1040.434,23.440,416.222,169.478,37.627,157.076
C00678=1040.428,23.190,416.238,169.476,37.626,157.076
C00679=1040.422,22.941,416.253,169.474,37.626,157.076
C00680=1040.416,22.692,416.269,169.472,37.625,157.076
C00681=1040.408,22.442,416.285,169.470,37.624,157.076
C00682=1040.402,22.193,416.302,169.469,37.623,157.076
C00683=1040.397,21.944,416.318,169.466,37.623,157.075
C00684=1040.390,21.694,416.333,169.464,37.622,157.075
C00685=1040.384,21.445,416.349,169.462,37.621,157.075
C00686=1040.377,21.196,416.365,169.460,37.621,157.075
C00687=1040.372,20.946,416.381,169.458,37.620,157.075
C00688=1040.365,20.697,416.396,169.456,37.619,157.075
C00689=1040.359,20.446,416.413,169.454,37.618,157.075
C00690=1040.352,20.197,416.428,169.452,37.618,157.074
C00691=1040.346,19.948,416.445,169.450,37.617,157.074
C00692=1040.340,19.698,416.460,169.448,37.617,157.074
C00693=1040.334,19.449,416.476,169.446,37.615,157.074
C00694=1040.327,19.200,416.491,169.444,37.615,157.074
C00695=1040.320,18.951,416.507,169.442,37.614,157.074
C00696=1040.315,18.701,416.523,169.440,37.614,157.073
C00697=1040.308,18.452,416.538,169.438,37.613,157.073
C00698=1040.302,18.203,416.555,169.436,37.613,157.073
C00699=1040.295,17.952,416.570,169.434,37.612,157.073
C00700=1040.288,17.703,416.586,169.432,37.611,157.073
C00701=1040.282,17.454,416.602,169.430,37.611,157.073
C00702=1040.276,17.204,416.617,169.427,37.610,157.073
C00703=1040.270,16.955,416.633,169.425,37.609,157.072
C00704=1040.264,16.705,416.648,169.423,37.608,157.072
C00705=1040.257,16.456,416.664,169.422,37.608,157.072
C00706=1040.251,16.207,416.680,169.420,37.607,157.072
C00707=1040.245,15.957,416.695,169.418,37.607,157.072
C00708=1040.238,15.708,416.710,169.416,37.606,157.072
C00709=1040.232,15.458,416.726,169.414,37.605,157.072
C00710=1040.226,15.209,416.742,169.411,37.604,157.071
C00711=1040.220,14.960,416.758,169.409,37.604,157.071
C00712=1040.213,14.710,416.773,169.407,37.603,157.071
C00713=1040.207,14.461,416.789,169.405,37.603,157.071
C00714=1040.201,14.211,416.804,169.403,37.602,157.071
C00715=1040.194,13.962,416.820,169.401,37.601,157.071
C00716=1040.188,13.712,416.835,169.399,37.601,157.071
C00717=1040.181,13.463,416.850,169.397,37.600,157.070
C00718=1040.175,13.214,416.865,169.395,37.600,157.070
C00719=1040.167,12.929,416.883,169.393,37.599,157.070
C00720=1040.160,12.643,416.901,169.390,37.598,157.070
C00721=1040.153,12.358,416.919,169.388,37.598,157.070
C00722=1040.146,12.072,416.936,169.385,37.597,157.070
C00723=1040.139,11.823,416.952,169.383,37.596,157.070
C00724=1040.133,11.573,416.967,169.381,37.595,157.069
C00725=1040.126,11.324,416.982,169.379,37.595,157.069
C00726=1040.120,11.075,416.997,169.377,37.594,157.069
C00727=1040.113,10.825,417.012,169.376,37.594,157.069
C00728=1040.106,10.576,417.028,169.374,37.594,157.069
C00729=1040.101,10.326,417.043,169.372,37.593,157.069
C00730=1040.094,10.077,417.059,169.369,37.593,157.069
C00731=1040.088,9.827,417.074,169.367,37.592,157.069
C00732=1040.081,9.578,417.089,169.365,37.591,157.068
C00733=1040.075,9.329,417.104,169.363,37.591,157.068
C00734=1040.068,9.079,417.119,169.361,37.590,157.068
C00735=1040.062,8.829,417.134,169.359,37.590,157.068
C00736=1040.055,8.580,417.150,169.357,37.589,157.068
C00737=1040.049,8.331,417.165,169.355,37.589,157.068
C00738=1040.042,8.081,417.180,169.353,37.588,157.068
C00739=1040.036,7.832,417.196,169.351,37.587,157.068
C00740=1040.030,7.582,417.211,169.348,37.587,157.067
C00741=1040.024,7.332,417.226,169.346,37.586,157.067
C00742=1040.017,7.083,417.241,169.344,37.586,157.067
C00743=1040.011,6.833,417.257,169.342,37.585,157.067
C00744=1040.004,6.584,417.272,169.340,37.584,157.067
C00745=1039.998,6.334,417.287,169.338,37.584,157.067
C00746=1039.991,6.085,417.302,169.336,37.583,157.067
C00747=1039.985,5.836,417.317,169.334,37.583,157.066
C00748=1039.979,5.587,417.332,169.332,37.582,157.066
C00749=1039.973,5.337,417.347,169.330,37.581,157.066
C00750=1039.966,5.087,417.362,169.328,37.581,157.066
C00751=1039.960,4.838,417.378,169.325,37.580,157.066
C00752=1039.954,4.588,417.393,169.323,37.580,157.066
C00753=1039.948,4.339,417.408,169.321,37.579,157.066
C00754=1039.941,4.089,417.423,169.319,37.579,157.066
C00755=1039.935,3.840,417.437,169.317,37.577,157.065
C00756=1039.929,3.591,417.453,169.315,37.577,157.065
C00757=1039.922,3.341,417.468,169.313,37.576,157.065
C00758=1039.916,3.092,417.483,169.311,37.576,157.065
C00759=1039.910,2.842,417.498,169.309,37.575,157.065
C00760=1039.903,2.592,417.513,169.306,37.574,157.065
C00761=1039.897,2.343,417.528,169.304,37.574,157.064
C00762=1039.891,2.094,417.542,169.302,37.573,157.064
C00763=1039.884,1.845,417.558,169.300,37.573,157.064
C00764=1039.878,1.595,417.573,169.298,37.572,157.064
C00765=1039.872,1.345,417.588,169.296,37.571,157.064
C00766=1039.865,1.096,417.603,169.294,37.571,157.064
C00767=1039.859,0.847,417.617,169.292,37.570,157.064
C00768=1039.854,0.597,417.633,169.290,37.570,157.064
C00769=1039.847,0.347,417.648,169.288,37.569,157.063
C00770=1039.841,0.097,417.663,169.285,37.569,157.063
C00771=1039.835,-0.152,417.678,169.283,37.568,157.063
C00772=1039.829,-0.401,417.692,169.281,37.567,157.063
C00773=1039.822,-0.651,417.707,169.279,37.567,157.063
C00774=1039.816,-0.901,417.722,169.277,37.566,157.063
C00775=1039.810,-1.150,417.737,169.275,37.566,157.063
C00776=1039.804,-1.398,417.752,169.273,37.565,157.063
C00777=1039.797,-1.648,417.767,169.271,37.564,157.062
C00778=1039.791,-1.898,417.782,169.269,37.564,157.062
C00779=1039.784,-2.147,417.797,169.267,37.563,157.062
C00780=1039.779,-2.396,417.812,169.265,37.563,157.062
C00781=1039.772,-2.646,417.827,169.262,37.562,157.062
C00782=1039.766,-2.896,417.841,169.260,37.561,157.062
C00783=1039.759,-3.179,417.858,169.258,37.561,157.062
C00784=1039.752,-3.463,417.875,169.256,37.560,157.061
C00785=1039.745,-3.746,417.891,169.253,37.560,157.061
C00786=1039.737,-4.030,417.909,169.251,37.559,157.061
C00787=1039.731,-4.279,417.923,169.249,37.559,157.061
C00788=1039.725,-4.529,417.937,169.247,37.558,157.061
C00789=1039.718,-4.779,417.952,169.245,37.557,157.061
C00790=1039.712,-5.028,417.967,169.243,37.557,157.061
C00791=1039.705,-5.277,417.981,169.240,37.556,157.061
C00792=1039.699,-5.527,417.996,169.238,37.556,157.061
C00793=1039.693,-5.776,418.011,169.235,37.556,157.060
C00794=1039.686,-6.026,418.024,169.233,37.555,157.060
C00795=1039.680,-6.275,418.039,169.231,37.555,157.060
C00796=1039.674,-6.525,418.054,169.229,37.554,157.060
C00797=1039.667,-6.774,418.069,169.227,37.553,157.060
C00798=1039.660,-7.024,418.083,169.225,37.553,157.060
C00799=1039.655,-7.273,418.097,169.223,37.553,157.060
C00800=1039.648,-7.523,418.112,169.221,37.552,157.060
C00801=1039.641,-7.772,418.126,169.219,37.552,157.059
C00802=1039.635,-8.021,418.141,169.217,37.551,157.059
C00803=1039.629,-8.272,418.155,169.214,37.550,157.059
C00804=1039.622,-8.521,418.170,169.212,37.551,157.059
C00805=1039.616,-8.770,418.184,169.210,37.550,157.059
C00806=1039.610,-9.020,418.199,169.208,37.549,157.059
C00807=1039.603,-9.270,418.213,169.205,37.549,157.059
C00808=1039.598,-9.519,418.227,169.203,37.548,157.059
C00809=1039.591,-9.768,418.242,169.201,37.548,157.059
C00810=1039.584,-10.018,418.256,169.199,37.548,157.059
C00811=1039.579,-10.267,418.271,169.197,37.547,157.058
C00812=1039.572,-10.517,418.285,169.195,37.546,157.058
C00813=1039.565,-10.767,418.299,169.193,37.546,157.058
C00814=1039.560,-11.016,418.314,169.191,37.545,157.058
C00815=1039.553,-11.265,418.329,169.188,37.545,157.058
C00816=1039.546,-11.515,418.342,169.186,37.544,157.058
C00817=1039.541,-11.764,418.357,169.184,37.544,157.058
C00818=1039.534,-12.014,418.372,169.182,37.544,157.058
C00819=1039.528,-12.263,418.385,169.180,37.543,157.057
C00820=1039.522,-12.513,418.400,169.177,37.542,157.057
C00821=1039.516,-12.763,418.414,169.175,37.542,157.057
C00822=1039.509,-13.012,418.428,169.173,37.541,157.057
C00823=1039.503,-13.261,418.443,169.171,37.541,157.057
C00824=1039.497,-13.511,418.457,169.169,37.541,157.057
C00825=1039.490,-13.760,418.471,169.167,37.540,157.057
C00826=1039.484,-14.011,418.486,169.165,37.540,157.057
C00827=1039.478,-14.260,418.500,169.162,37.539,157.057
C00828=1039.471,-14.510,418.514,169.160,37.538,157.056
C00829=1039.466,-14.758,418.528,169.158,37.538,157.056
C00830=1039.459,-15.008,418.543,169.156,37.538,157.056
C00831=1039.453,-15.257,418.557,169.153,37.537,157.056
C00832=1039.447,-15.507,418.572,169.151,37.537,157.056
C00833=1039.440,-15.757,418.585,169.149,37.536,157.056
C00834=1039.434,-16.007,418.599,169.147,37.536,157.056
C00835=1039.427,-16.256,418.613,169.145,37.536,157.056
C00836=1039.421,-16.505,418.627,169.143,37.535,157.056
C00837=1039.415,-16.755,418.642,169.141,37.535,157.056
C00838=1039.408,-17.004,418.655,169.138,37.534,157.055
C00839=1039.402,-17.254,418.670,169.136,37.534,157.055
C00840=1039.395,-17.504,418.684,169.134,37.534,157.055
C00841=1039.389,-17.753,418.697,169.131,37.533,157.055
C00842=1039.383,-18.003,418.712,169.129,37.533,157.055
C00843=1039.376,-18.252,418.725,169.127,37.532,157.055
C00844=1039.370,-18.502,418.740,169.125,37.532,157.055
C00845=1039.364,-18.751,418.753,169.123,37.532,157.055
C00846=1039.357,-19.001,418.767,169.120,37.531,157.055
C00847=1039.350,-19.282,418.783,169.118,37.531,157.055
C00848=1039.342,-19.564,418.799,169.116,37.530,157.054
C00849=1039.336,-19.847,418.815,169.113,37.530,157.054
C00850=1039.329,-20.128,418.830,169.111,37.529,157.054
C00851=1039.322,-20.378,418.844,169.109,37.529,157.054
C00852=1039.316,-20.627,418.857,169.106,37.529,157.054
C00853=1039.310,-20.877,418.872,169.104,37.528,157.054
C00854=1039.303,-21.126,418.886,169.101,37.528,157.054
C00855=1039.297,-21.376,418.899,169.099,37.528,157.054
C00856=1039.291,-21.625,418.913,169.097,37.527,157.054
C00857=1039.284,-21.875,418.927,169.095,37.526,157.053
C00858=1039.279,-22.124,418.941,169.092,37.527,157.053
C00859=1039.272,-22.374,418.955,169.090,37.526,157.053
C00860=1039.265,-22.623,418.969,169.088,37.525,157.053
C00861=1039.259,-22.873,418.983,169.086,37.525,157.053
C00862=1039.253,-23.122,418.996,169.084,37.525,157.053
C00863=1039.246,-23.372,419.010,169.082,37.524,157.053
C00864=1039.241,-23.622,419.024,169.080,37.524,157.053
C00865=1039.234,-23.871,419.038,169.077,37.524,157.053
C00866=1039.227,-24.121,419.051,169.075,37.523,157.053
C00867=1039.222,-24.370,419.065,169.073,37.523,157.053
C00868=1039.215,-24.620,419.079,169.071,37.523,157.053
C00869=1039.210,-24.870,419.093,169.068,37.522,157.052
C00870=1039.203,-25.118,419.107,169.066,37.521,157.052
C00871=1039.196,-25.368,419.120,169.063,37.521,157.052
C00872=1039.191,-25.618,419.134,169.061,37.521,157.052
C00873=1039.184,-25.868,419.148,169.059,37.520,157.052
C00874=1039.178,-26.117,419.161,169.057,37.520,157.052
C00875=1039.172,-26.367,419.175,169.055,37.520,157.052
C00876=1039.165,-26.617,419.189,169.053,37.519,157.052
C00877=1039.159,-26.866,419.202,169.050,37.519,157.052
C00878=1039.154,-27.115,419.216,169.048,37.519,157.052
C00879=1039.147,-27.365,419.230,169.046,37.518,157.051
C00880=1039.140,-27.614,419.243,169.044,37.518,157.051
C00881=1039.134,-27.864,419.257,169.042,37.518,157.051
C00882=1039.127,-28.113,419.270,169.039,37.518,157.051
C00883=1039.121,-28.363,419.284,169.037,37.517,157.051
C00884=1039.114,-28.613,419.297,169.035,37.517,157.051
C00885=1039.108,-28.862,419.311,169.032,37.516,157.051
C00886=1039.101,-29.112,419.324,169.029,37.517,157.051
C00887=1039.095,-29.361,419.337,169.027,37.516,157.051
C00888=1039.090,-29.611,419.351,169.025,37.516,157.051
C00889=1039.083,-29.861,419.364,169.023,37.515,157.051
C00890=1039.077,-30.110,419.378,169.021,37.515,157.051
C00891=1039.071,-30.360,419.391,169.018,37.515,157.051
C00892=1039.064,-30.610,419.404,169.016,37.514,157.050
C00893=1039.058,-30.859,419.418,169.014,37.514,157.050
C00894=1039.051,-31.108,419.431,169.012,37.514,157.050
C00895=1039.045,-31.358,419.445,169.009,37.514,157.050
C00896=1039.038,-31.607,419.458,169.007,37.513,157.050
C00897=1039.032,-31.857,419.471,169.005,37.513,157.050
C00898=1039.025,-32.107,419.485,169.003,37.513,157.050
C00899=1039.019,-32.356,419.498,169.001,37.513,157.050
C00900=1039.013,-32.605,419.511,168.998,37.512,157.050
C00901=1039.008,-32.855,419.524,168.996,37.512,157.050
C00902=1039.001,-33.105,419.538,168.994,37.512,157.050
C00903=1038.995,-33.355,419.551,168.992,37.512,157.050
C00904=1038.989,-33.604,419.565,168.988,37.511,157.050
C00905=1038.982,-33.853,419.578,168.986,37.511,157.050
C00906=1038.975,-34.103,419.592,168.984,37.511,157.049
C00907=1038.970,-34.353,419.604,168.982,37.511,157.049
C00908=1038.963,-34.602,419.617,168.979,37.510,157.049
C00909=1038.957,-34.851,419.631,168.977,37.510,157.049
C00910=1038.950,-35.101,419.644,168.975,37.510,157.049
C00911=1038.944,-35.382,419.658,168.972,37.509,157.049
C00912=1038.937,-35.663,419.674,168.970,37.509,157.049
C00913=1038.929,-35.945,419.689,168.967,37.508,157.049
C00914=1038.922,-36.226,419.704,168.965,37.508,157.049
C00915=1038.916,-36.476,419.717,168.963,37.508,157.049
C00916=1038.910,-36.725,419.730,168.960,37.508,157.049
C00917=1038.904,-36.974,419.743,168.958,37.507,157.049
C00918=1038.898,-37.223,419.757,168.956,37.507,157.049
C00919=1038.891,-37.474,419.770,168.954,37.507,157.048
C00920=1038.885,-37.723,419.783,168.951,37.507,157.048
C00921=1038.879,-37.973,419.796,168.949,37.506,157.048
C00922=1038.873,-38.222,419.809,168.947,37.506,157.048
C00923=1038.867,-38.472,419.822,168.944,37.506,157.048
C00924=1038.860,-38.722,419.836,168.941,37.506,157.048
C00925=1038.854,-38.972,419.848,168.939,37.505,157.048
C00926=1038.848,-39.221,419.861,168.937,37.505,157.048
C00927=1038.841,-39.470,419.874,168.934,37.505,157.048
C00928=1038.835,-39.720,419.887,168.932,37.505,157.048
C00929=1038.828,-39.970,419.900,168.930,37.505,157.048
C00930=1038.822,-40.220,419.913,168.928,37.504,157.048
C00931=1038.816,-40.469,419.926,168.925,37.504,157.048
C00932=1038.809,-40.718,419.939,168.923,37.504,157.048
C00933=1038.803,-40.968,419.951,168.921,37.504,157.047
C00934=1038.797,-41.217,419.965,168.918,37.504,157.047
C00935=1038.790,-41.467,419.977,168.916,37.504,157.047
C00936=1038.784,-41.717,419.991,168.914,37.503,157.047
C00937=1038.778,-41.966,420.003,168.911,37.503,157.047
C00938=1038.771,-42.216,420.016,168.909,37.503,157.047
C00939=1038.765,-42.465,420.029,168.907,37.503,157.047
C00940=1038.759,-42.715,420.042,168.905,37.503,157.047
C00941=1038.753,-42.964,420.054,168.902,37.502,157.047
C00942=1038.746,-43.214,420.067,168.900,37.502,157.047
C00943=1038.740,-43.464,420.080,168.898,37.502,157.047
C00944=1038.734,-43.713,420.093,168.895,37.502,157.047
C00945=1038.727,-43.963,420.105,168.893,37.502,157.047
C00946=1038.721,-44.212,420.118,168.891,37.502,157.047
C00947=1038.715,-44.462,420.131,168.887,37.501,157.047
C00948=1038.709,-44.712,420.144,168.885,37.501,157.047
C00949=1038.703,-44.961,420.157,168.883,37.501,157.047
C00950=1038.696,-45.211,420.169,168.880,37.501,157.047
C00951=1038.690,-45.460,420.182,168.878,37.501,157.046
C00952=1038.684,-45.710,420.195,168.876,37.501,157.046
C00953=1038.678,-45.959,420.208,168.874,37.500,157.046
C00954=1038.671,-46.209,420.220,168.871,37.500,157.046
C00955=1038.665,-46.459,420.232,168.869,37.501,157.046
C00956=1038.659,-46.708,420.246,168.867,37.500,157.046
C00957=1038.652,-46.958,420.258,168.864,37.500,157.046
C00958=1038.646,-47.208,420.271,168.862,37.500,157.046
C00959=1038.640,-47.457,420.284,168.860,37.499,157.046
C00960=1038.634,-47.707,420.296,168.857,37.500,157.046
C00961=1038.627,-47.957,420.308,168.855,37.500,157.046
C00962=1038.621,-48.206,420.322,168.853,37.499,157.046
C00963=1038.615,-48.456,420.334,168.850,37.499,157.046
C00964=1038.609,-48.706,420.347,168.848,37.499,157.046
C00965=1038.602,-48.955,420.359,168.846,37.499,157.046
C00966=1038.596,-49.205,420.372,168.843,37.499,157.046
C00967=1038.591,-49.454,420.384,168.841,37.499,157.046
C00968=1038.585,-49.704,420.397,168.839,37.499,157.046
C00969=1038.578,-49.953,420.409,168.836,37.498,157.046
C00970=1038.572,-50.203,420.422,168.834,37.498,157.046
C00971=1038.566,-50.453,420.434,168.832,37.498,157.045
C00972=1038.560,-50.702,420.446,168.829,37.498,157.045
C00973=1038.553,-50.951,420.460,168.827,37.498,157.045
C00974=1038.547,-51.201,420.472,168.824,37.498,157.045
C00975=1038.540,-51.483,420.485,168.821,37.498,157.045
C00976=1038.532,-51.764,420.499,168.818,37.498,157.045
C00977=1038.525,-52.046,420.513,168.815,37.498,157.045
C00978=1038.517,-52.328,420.527,168.813,37.498,157.045
C00979=1038.511,-52.577,420.539,168.810,37.498,157.045
C00980=1038.505,-52.827,420.552,168.808,37.498,157.045
C00981=1038.498,-53.077,420.564,168.805,37.498,157.045
C00982=1038.492,-53.326,420.576,168.803,37.498,157.045
C00983=1038.486,-53.575,420.588,168.801,37.498,157.045
C00984=1038.479,-53.825,420.600,168.798,37.498,157.045
C00985=1038.473,-54.075,420.612,168.796,37.498,157.045
C00986=1038.467,-54.324,420.624,168.793,37.498,157.045
C00987=1038.460,-54.574,420.636,168.791,37.498,157.045
C00988=1038.454,-54.824,420.649,168.789,37.498,157.045
C00989=1038.448,-55.073,420.661,168.786,37.498,157.045
C00990=1038.441,-55.323,420.673,168.784,37.498,157.045
C00991=1038.435,-55.573,420.685,168.781,37.498,157.045
C00992=1038.428,-55.822,420.697,168.779,37.498,157.045
C00993=1038.422,-56.072,420.709,168.777,37.498,157.045
C00994=1038.416,-56.322,420.722,168.774,37.498,157.045
C00995=1038.409,-56.571,420.734,168.772,37.498,157.045
C00996=1038.403,-56.821,420.746,168.769,37.499,157.045
C00997=1038.397,-57.070,420.758,168.767,37.499,157.045
C00998=1038.391,-57.320,420.770,168.765,37.499,157.045
C00999=1038.384,-57.569,420.782,168.762,37.499,157.045
C01000=1038.378,-57.819,420.794,168.760,37.499,157.045
C01001=1038.371,-58.069,420.806,168.757,37.499,157.045
C01002=1038.365,-58.318,420.818,168.755,37.498,157.045
C01003=1038.359,-58.568,420.831,168.752,37.498,157.045
C01004=1038.353,-58.817,420.843,168.750,37.498,157.045
C01005=1038.346,-59.067,420.854,168.748,37.498,157.045
C01006=1038.341,-59.317,420.866,168.745,37.499,157.045
C01007=1038.334,-59.567,420.878,168.743,37.499,157.045
C01008=1038.327,-59.816,420.890,168.740,37.499,157.045
C01009=1038.321,-60.066,420.903,168.738,37.499,157.045
C01010=1038.315,-60.315,420.914,168.735,37.499,157.045
C01011=1038.309,-60.565,420.926,168.733,37.499,157.045
C01012=1038.303,-60.815,420.939,168.731,37.499,157.044
C01013=1038.296,-61.065,420.950,168.728,37.499,157.044
C01014=1038.290,-61.314,420.962,168.726,37.499,157.044
C01015=1038.284,-61.563,420.974,168.723,37.499,157.044
C01016=1038.278,-61.813,420.986,168.721,37.499,157.044
C01017=1038.271,-62.063,420.998,168.718,37.499,157.044
C01018=1038.265,-62.313,421.009,168.716,37.499,157.044
C01019=1038.259,-62.563,421.022,168.714,37.499,157.044
C01020=1038.253,-62.812,421.034,168.711,37.499,157.044
C01021=1038.246,-63.061,421.046,168.709,37.499,157.044
C01022=1038.241,-63.312,421.057,168.706,37.500,157.044
C01023=1038.234,-63.561,421.069,168.704,37.500,157.044
C01024=1038.228,-63.810,421.081,168.701,37.500,157.044
C01025=1038.221,-64.060,421.093,168.699,37.500,157.044
C01026=1038.216,-64.310,421.105,168.697,37.500,157.044
C01027=1038.210,-64.559,421.116,168.694,37.500,157.044
C01028=1038.203,-64.809,421.128,168.692,37.500,157.044
C01029=1038.197,-65.059,421.140,168.689,37.500,157.044
C01030=1038.191,-65.309,421.152,168.687,37.500,157.044
C01031=1038.185,-65.558,421.164,168.684,37.500,157.044
C01032=1038.178,-65.808,421.175,168.682,37.500,157.044
C01033=1038.172,-66.058,421.187,168.679,37.500,157.044
C01034=1038.166,-66.306,421.199,168.677,37.500,157.044
C01035=1038.160,-66.557,421.210,168.675,37.500,157.044
C01036=1038.153,-66.806,421.222,168.672,37.500,157.044
C01037=1038.148,-67.055,421.234,168.670,37.500,157.044
C01038=1038.142,-67.306,421.246,168.667,37.501,157.044
C01039=1038.135,-67.588,421.259,168.664,37.501,157.044
C01040=1038.127,-67.871,421.273,168.662,37.501,157.044
C01041=1038.121,-68.154,421.286,168.659,37.501,157.044
C01042=1038.114,-68.436,421.299,168.656,37.501,157.044
C01043=1038.108,-68.687,421.310,168.654,37.501,157.044
C01044=1038.101,-68.935,421.322,168.651,37.501,157.044
C01045=1038.096,-69.185,421.334,168.649,37.501,157.044
C01046=1038.089,-69.436,421.345,168.646,37.501,157.044
C01047=1038.083,-69.684,421.357,168.644,37.501,157.044
C01048=1038.077,-69.935,421.368,168.641,37.501,157.044
C01049=1038.072,-70.184,421.380,168.639,37.501,157.044
C01050=1038.065,-70.434,421.392,168.636,37.501,157.044
C01051=1038.059,-70.684,421.404,168.634,37.501,157.044
C01052=1038.053,-70.933,421.415,168.631,37.502,157.044
C01053=1038.047,-71.183,421.427,168.629,37.502,157.044
C01054=1038.041,-71.432,421.438,168.627,37.502,157.044
C01055=1038.035,-71.682,421.450,168.624,37.502,157.044
C01056=1038.029,-71.931,421.461,168.622,37.502,157.044
C01057=1038.022,-72.181,421.473,168.619,37.502,157.044
C01058=1038.017,-72.431,421.484,168.617,37.503,157.044
C01059=1038.011,-72.681,421.495,168.614,37.503,157.044
C01060=1038.005,-72.930,421.507,168.612,37.503,157.044
C01061=1037.998,-73.180,421.518,168.609,37.503,157.044
C01062=1037.992,-73.430,421.530,168.607,37.503,157.044
C01063=1037.987,-73.679,421.542,168.604,37.503,157.044
C01064=1037.980,-73.930,421.553,168.602,37.503,157.044
C01065=1037.974,-74.179,421.565,168.599,37.503,157.044
C01066=1037.968,-74.429,421.576,168.597,37.503,157.044
C01067=1037.962,-74.678,421.587,168.594,37.504,157.044
C01068=1037.956,-74.928,421.599,168.592,37.504,157.044
C01069=1037.950,-75.177,421.610,168.589,37.504,157.044
C01070=1037.944,-75.427,421.621,168.587,37.504,157.044
C01071=1037.938,-75.676,421.632,168.584,37.505,157.044
C01072=1037.931,-75.927,421.644,168.582,37.505,157.044
C01073=1037.925,-76.176,421.654,168.579,37.505,157.044
C01074=1037.918,-76.426,421.665,168.577,37.505,157.044
C01075=1037.912,-76.675,421.677,168.574,37.506,157.044
C01076=1037.906,-76.925,421.688,168.572,37.506,157.044
C01077=1037.900,-77.174,421.699,168.569,37.506,157.044
C01078=1037.894,-77.425,421.710,168.567,37.506,157.044
C01079=1037.888,-77.674,421.722,168.564,37.507,157.044
C01080=1037.882,-77.924,421.733,168.562,37.507,157.044
C01081=1037.876,-78.173,421.744,168.559,37.507,157.044
C01082=1037.869,-78.423,421.755,168.556,37.507,157.044
C01083=1037.864,-78.673,421.766,168.554,37.507,157.044
C01084=1037.857,-78.923,421.777,168.551,37.508,157.044
C01085=1037.851,-79.172,421.789,168.549,37.508,157.044
C01086=1037.844,-79.422,421.799,168.546,37.508,157.044
C01087=1037.838,-79.671,421.810,168.544,37.508,157.044
C01088=1037.833,-79.921,421.821,168.541,37.508,157.044
C01089=1037.826,-80.171,421.832,168.539,37.509,157.044
C01090=1037.821,-80.420,421.843,168.536,37.509,157.044
C01091=1037.814,-80.670,421.854,168.534,37.510,157.044
C01092=1037.808,-80.920,421.865,168.531,37.510,157.044
C01093=1037.802,-81.170,421.876,168.528,37.510,157.044
C01094=1037.795,-81.419,421.886,168.526,37.511,157.044
C01095=1037.789,-81.669,421.898,168.523,37.511,157.044
C01096=1037.783,-81.919,421.908,168.521,37.512,157.044
C01097=1037.776,-82.169,421.919,168.518,37.512,157.044
C01098=1037.770,-82.418,421.930,168.516,37.512,157.044
C01099=1037.764,-82.668,421.941,168.513,37.512,157.044
C01100=1037.757,-82.918,421.952,168.510,37.513,157.045
C01101=1037.752,-83.167,421.962,168.508,37.513,157.045
C01102=1037.745,-83.417,421.974,168.505,37.514,157.045
C01103=1037.738,-83.701,421.986,168.502,37.514,157.045
C01104=1037.731,-83.987,421.999,168.499,37.515,157.045
C01105=1037.724,-84.271,422.011,168.496,37.515,157.045
C01106=1037.717,-84.557,422.023,168.494,37.516,157.045
C01107=1037.711,-84.806,422.034,168.492,37.516,157.045
C01108=1037.704,-85.056,422.044,168.489,37.516,157.045
C01109=1037.698,-85.306,422.055,168.487,37.516,157.045
C01110=1037.692,-85.555,422.065,168.484,37.517,157.045
C01111=1037.685,-85.805,422.077,168.481,37.517,157.045
C01112=1037.680,-86.054,422.088,168.479,37.518,157.045
C01113=1037.674,-86.304,422.097,168.476,37.518,157.045
C01114=1037.667,-86.554,422.108,168.474,37.519,157.045
C01115=1037.661,-86.804,422.119,168.471,37.519,157.045
C01116=1037.655,-87.053,422.130,168.469,37.520,157.045
C01117=1037.649,-87.303,422.141,168.466,37.520,157.045
C01118=1037.643,-87.553,422.152,168.463,37.520,157.045
C01119=1037.637,-87.803,422.161,168.461,37.520,157.045
C01120=1037.630,-88.053,422.173,168.458,37.521,157.045
C01121=1037.624,-88.302,422.183,168.456,37.521,157.045
C01122=1037.618,-88.551,422.194,168.453,37.522,157.045
C01123=1037.612,-88.801,422.205,168.450,37.523,157.045
C01124=1037.606,-89.051,422.214,168.448,37.523,157.045
C01125=1037.600,-89.301,422.225,168.445,37.523,157.046
C01126=1037.593,-89.550,422.236,168.443,37.524,157.046
C01127=1037.587,-89.800,422.247,168.440,37.524,157.046
C01128=1037.581,-90.050,422.258,168.437,37.524,157.046
C01129=1037.575,-90.300,422.267,168.435,37.525,157.046
C01130=1037.569,-90.549,422.278,168.432,37.525,157.046
C01131=1037.563,-90.798,422.288,168.430,37.526,157.046
C01132=1037.557,-91.049,422.299,168.427,37.526,157.046
C01133=1037.551,-91.299,422.310,168.424,37.527,157.046
C01134=1037.545,-91.548,422.320,168.422,37.527,157.046
C01135=1037.539,-91.797,422.331,168.420,37.527,157.046
C01136=1037.532,-92.048,422.341,168.418,37.528,157.046
C01137=1037.526,-92.297,422.352,168.415,37.528,157.046
C01138=1037.521,-92.547,422.363,168.412,37.529,157.046
C01139=1037.515,-92.796,422.372,168.410,37.529,157.046
C01140=1037.509,-93.046,422.383,168.407,37.530,157.046
C01141=1037.503,-93.296,422.393,168.404,37.530,157.046
C01142=1037.496,-93.546,422.404,168.402,37.531,157.046
C01143=1037.490,-93.795,422.414,168.399,37.531,157.046
C01144=1037.484,-94.045,422.424,168.397,37.531,157.046
C01145=1037.479,-94.295,422.435,168.394,37.532,157.046
C01146=1037.472,-94.544,422.446,168.391,37.532,157.046
C01147=1037.467,-94.794,422.456,168.389,37.533,157.047
C01148=1037.460,-95.044,422.466,168.386,37.533,157.047
C01149=1037.454,-95.294,422.477,168.384,37.534,157.047
C01150=1037.448,-95.543,422.487,168.381,37.534,157.047
C01151=1037.442,-95.793,422.497,168.378,37.535,157.047
C01152=1037.436,-96.042,422.507,168.376,37.535,157.047
C01153=1037.430,-96.292,422.518,168.373,37.535,157.047
C01154=1037.425,-96.542,422.528,168.371,37.536,157.047
C01155=1037.418,-96.791,422.539,168.368,37.537,157.047
C01156=1037.413,-97.041,422.549,168.365,37.537,157.047
C01157=1037.406,-97.292,422.559,168.363,37.538,157.047
C01158=1037.400,-97.541,422.570,168.361,37.538,157.047
C01159=1037.394,-97.791,422.579,168.357,37.538,157.047
C01160=1037.388,-98.040,422.589,168.356,37.539,157.047
C01161=1037.382,-98.290,422.600,168.353,37.540,157.047
C01162=1037.376,-98.540,422.610,168.350,37.541,157.047
C01163=1037.370,-98.789,422.619,168.348,37.541,157.047
C01164=1037.364,-99.040,422.630,168.345,37.541,157.048
C01165=1037.358,-99.289,422.640,168.342,37.542,157.048
C01166=1037.351,-99.539,422.650,168.340,37.543,157.048
C01167=1037.345,-99.826,422.661,168.337,37.544,157.048
C01168=1037.337,-100.113,422.673,168.334,37.544,157.048
C01169=1037.330,-100.400,422.684,168.331,37.545,157.048
C01170=1037.323,-100.688,422.696,168.327,37.546,157.048
C01171=1037.317,-100.938,422.706,168.325,37.546,157.048
C01172=1037.311,-101.187,422.716,168.322,37.547,157.048
C01173=1037.305,-101.437,422.726,168.319,37.547,157.048
C01174=1037.299,-101.687,422.736,168.317,37.548,157.048
C01175=1037.293,-101.936,422.746,168.315,37.549,157.048
C01176=1037.286,-102.186,422.756,168.312,37.550,157.049
C01177=1037.281,-102.436,422.766,168.310,37.550,157.049
C01178=1037.275,-102.686,422.775,168.307,37.550,157.049
C01179=1037.268,-102.935,422.786,168.304,37.551,157.049
C01180=1037.262,-103.185,422.795,168.302,37.552,157.049
C01181=1037.257,-103.435,422.805,168.299,37.553,157.049
C01182=1037.251,-103.684,422.815,168.296,37.553,157.049
C01183=1037.244,-103.934,422.825,168.294,37.553,157.049
C01184=1037.238,-104.183,422.835,168.291,37.554,157.049
C01185=1037.233,-104.434,422.845,168.288,37.555,157.049
C01186=1037.226,-104.683,422.855,168.286,37.556,157.049
C01187=1037.220,-104.933,422.864,168.283,37.556,157.049
C01188=1037.214,-105.182,422.874,168.280,37.557,157.049
C01189=1037.208,-105.432,422.885,168.278,37.558,157.050
C01190=1037.202,-105.682,422.894,168.276,37.558,157.050
C01191=1037.196,-105.932,422.904,168.273,37.559,157.050
C01192=1037.190,-106.182,422.913,168.271,37.559,157.050
C01193=1037.184,-106.432,422.923,168.268,37.560,157.050
C01194=1037.178,-106.682,422.933,168.265,37.561,157.050
C01195=1037.172,-106.931,422.943,168.263,37.561,157.050
C01196=1037.166,-107.181,422.953,168.260,37.562,157.050
C01197=1037.159,-107.430,422.962,168.257,37.563,157.050
C01198=1037.154,-107.680,422.972,168.255,37.564,157.050
C01199=1037.148,-107.929,422.981,168.252,37.564,157.050
C01200=1037.141,-108.179,422.991,168.249,37.565,157.050
C01201=1037.136,-108.429,423.001,168.246,37.566,157.051
C01202=1037.130,-108.679,423.011,168.244,37.567,157.051
C01203=1037.124,-108.929,423.020,168.241,37.567,157.051
C01204=1037.117,-109.179,423.030,168.238,37.568,157.051
C01205=1037.111,-109.428,423.039,168.237,37.569,157.051
C01206=1037.105,-109.678,423.049,168.234,37.570,157.051
C01207=1037.099,-109.928,423.058,168.231,37.570,157.051
C01208=1037.093,-110.177,423.068,168.228,37.571,157.051
C01209=1037.087,-110.427,423.077,168.226,37.572,157.051
C01210=1037.081,-110.677,423.087,168.223,37.573,157.051
C01211=1037.075,-110.927,423.096,168.220,37.573,157.051
C01212=1037.069,-111.176,423.106,168.218,37.574,157.052
C01213=1037.063,-111.426,423.115,168.215,37.575,157.052
C01214=1037.056,-111.676,423.125,168.212,37.576,157.052
C01215=1037.051,-111.925,423.134,168.209,37.577,157.052
C01216=1037.045,-112.175,423.144,168.207,37.578,157.052
C01217=1037.038,-112.425,423.153,168.205,37.578,157.052
C01218=1037.033,-112.675,423.162,168.202,37.579,157.052
C01219=1037.026,-112.925,423.172,168.200,37.580,157.052
C01220=1037.020,-113.175,423.181,168.197,37.581,157.052
C01221=1037.015,-113.424,423.191,168.194,37.581,157.053
C01222=1037.008,-113.674,423.200,168.191,37.582,157.053
C01223=1037.002,-113.923,423.210,168.189,37.583,157.053
C01224=1036.997,-114.173,423.220,168.186,37.583,157.053
C01225=1036.990,-114.424,423.228,168.183,37.584,157.053
C01226=1036.985,-114.673,423.237,168.181,37.586,157.053
C01227=1036.979,-114.922,423.247,168.178,37.586,157.053
C01228=1036.972,-115.172,423.256,168.175,37.587,157.053
C01229=1036.966,-115.422,423.266,168.173,37.588,157.053
C01230=1036.960,-115.672,423.275,168.171,37.589,157.054
C01231=1036.954,-115.958,423.285,168.167,37.590,157.054
C01232=1036.947,-116.245,423.296,168.164,37.591,157.054
C01233=1036.940,-116.531,423.306,168.161,37.592,157.054
C01234=1036.933,-116.818,423.317,168.158,37.593,157.054
C01235=1036.927,-117.068,423.327,168.155,37.594,157.054
C01236=1036.920,-117.317,423.336,168.153,37.594,157.054
C01237=1036.915,-117.567,423.344,168.150,37.595,157.054
C01238=1036.909,-117.817,423.354,168.147,37.596,157.054
C01239=1036.903,-118.066,423.364,168.145,37.597,157.055
C01240=1036.897,-118.316,423.373,168.143,37.598,157.055
C01241=1036.891,-118.566,423.382,168.140,37.599,157.055
C01242=1036.885,-118.816,423.391,168.137,37.600,157.055
C01243=1036.878,-119.065,423.400,168.134,37.601,157.055
C01244=1036.873,-119.315,423.409,168.132,37.602,157.055
C01245=1036.867,-119.565,423.418,168.129,37.602,157.055
C01246=1036.861,-119.815,423.427,168.126,37.603,157.055
C01247=1036.855,-120.064,423.436,168.123,37.605,157.056
C01248=1036.849,-120.314,423.446,168.121,37.605,157.056
C01249=1036.843,-120.564,423.454,168.119,37.606,157.056
C01250=1036.837,-120.813,423.463,168.116,37.607,157.056
C01251=1036.831,-121.064,423.472,168.113,37.608,157.056
C01252=1036.825,-121.314,423.482,168.111,37.609,157.056
C01253=1036.819,-121.563,423.491,168.108,37.610,157.056
C01254=1036.813,-121.813,423.499,168.105,37.611,157.057
C01255=1036.807,-122.063,423.509,168.102,37.612,157.057
C01256=1036.801,-122.312,423.517,168.100,37.613,157.057
C01257=1036.795,-122.562,423.527,168.097,37.613,157.057
C01258=1036.789,-122.812,423.536,168.094,37.615,157.057
C01259=1036.783,-123.061,423.544,168.092,37.615,157.057
C01260=1036.777,-123.312,423.553,168.089,37.616,157.057
C01261=1036.772,-123.561,423.562,168.087,37.618,157.057
C01262=1036.766,-123.811,423.571,168.084,37.618,157.057
C01263=1036.759,-124.061,423.580,168.081,37.619,157.058
C01264=1036.753,-124.310,423.589,168.078,37.621,157.058
C01265=1036.747,-124.560,423.598,168.076,37.621,157.058
C01266=1036.742,-124.810,423.607,168.073,37.623,157.058
C01267=1036.735,-125.060,423.615,168.070,37.623,157.058
C01268=1036.729,-125.310,423.624,168.067,37.624,157.058
C01269=1036.724,-125.559,423.633,168.066,37.626,157.058
C01270=1036.717,-125.809,423.642,168.063,37.626,157.059
C01271=1036.712,-126.059,423.650,168.060,37.628,157.059
C01272=1036.705,-126.309,423.659,168.057,37.628,157.059
C01273=1036.699,-126.559,423.668,168.054,37.630,157.059
C01274=1036.694,-126.808,423.677,168.052,37.631,157.059
C01275=1036.687,-127.058,423.686,168.049,37.631,157.059
C01276=1036.682,-127.308,423.694,168.046,37.633,157.059
C01277=1036.676,-127.558,423.703,168.044,37.634,157.060
C01278=1036.669,-127.807,423.712,168.041,37.635,157.060
C01279=1036.664,-128.056,423.720,168.039,37.636,157.060
C01280=1036.660,-128.306,423.730,168.036,37.636,157.060
C01281=1036.656,-128.556,423.741,168.034,37.636,157.060
C01282=1036.653,-128.806,423.752,168.032,37.635,157.060
C01283=1036.650,-129.056,423.763,168.029,37.634,157.059
C01284=1036.649,-129.306,423.775,168.027,37.632,157.059
C01285=1036.647,-129.556,423.788,168.025,37.630,157.059
C01286=1036.647,-129.805,423.801,168.024,37.627,157.058
C01287=1036.648,-130.056,423.816,168.021,37.625,157.058
C01288=1036.649,-130.305,423.830,168.020,37.621,157.057
C01289=1036.651,-130.555,423.844,168.018,37.618,157.057
C01290=1036.653,-130.805,423.860,168.017,37.613,157.056
C01291=1036.657,-131.056,423.876,168.016,37.608,157.055
C01292=1036.661,-131.306,423.893,168.014,37.603,157.054
C01293=1036.666,-131.556,423.911,168.014,37.598,157.053
C01294=1036.673,-131.806,423.929,168.012,37.591,157.052
C01295=1036.335,-131.830,423.655,167.964,37.802,157.087
C01296=1036.329,-131.581,423.637,167.965,37.808,157.088
C01297=1036.324,-131.330,423.619,167.966,37.814,157.089
C01298=1036.319,-131.081,423.602,167.968,37.819,157.090
C01299=1036.317,-130.830,423.586,167.969,37.824,157.091
C01300=1036.314,-130.580,423.570,167.970,37.828,157.091
C01301=1036.311,-130.330,423.555,167.971,37.832,157.092
C01302=1036.310,-130.080,423.541,167.974,37.836,157.093
C01303=1036.310,-129.830,423.527,167.975,37.839,157.093
C01304=1036.310,-129.580,423.513,167.977,37.841,157.093
C01305=1036.311,-129.331,423.501,167.979,37.843,157.094
C01306=1036.313,-129.081,423.489,167.981,37.845,157.094
C01307=1036.315,-128.830,423.477,167.983,37.846,157.094
C01308=1036.319,-128.580,423.466,167.985,37.847,157.095
C01309=1036.322,-128.330,423.455,167.987,37.847,157.095
C01310=1036.327,-128.081,423.446,167.991,37.846,157.095
C01311=1036.332,-127.831,423.437,167.993,37.846,157.095
C01312=1036.338,-127.582,423.428,167.995,37.845,157.094
C01313=1036.344,-127.332,423.420,167.998,37.843,157.094
C01314=1036.349,-127.082,423.411,168.001,37.843,157.094
C01315=1036.356,-126.833,423.402,168.004,37.841,157.094
C01316=1036.362,-126.583,423.394,168.007,37.841,157.094
C01317=1036.368,-126.333,423.384,168.009,37.839,157.094
C01318=1036.373,-126.084,423.376,168.012,37.838,157.094
C01319=1036.380,-125.834,423.367,168.014,37.837,157.093
C01320=1036.386,-125.584,423.358,168.017,37.836,157.093
C01321=1036.392,-125.334,423.350,168.020,37.835,157.093
C01322=1036.398,-125.084,423.341,168.022,37.834,157.093
C01323=1036.403,-124.835,423.332,168.025,37.833,157.093
C01324=1036.410,-124.585,423.324,168.028,37.832,157.093
C01325=1036.415,-124.336,423.314,168.031,37.831,157.093
C01326=1036.421,-124.085,423.306,168.034,37.830,157.092
C01327=1036.427,-123.835,423.296,168.036,37.829,157.092
C01328=1036.433,-123.586,423.288,168.038,37.827,157.092
C01329=1036.440,-123.336,423.278,168.041,37.827,157.092
C01330=1036.445,-123.087,423.270,168.044,37.826,157.092
C01331=1036.451,-122.837,423.260,168.046,37.824,157.092
C01332=1036.457,-122.586,423.252,168.049,37.824,157.092
C01333=1036.463,-122.338,423.243,168.052,37.823,157.092
C01334=1036.469,-122.087,423.234,168.055,37.822,157.091
C01335=1036.475,-121.837,423.225,168.058,37.821,157.091
C01336=1036.481,-121.588,423.216,168.060,37.820,157.091
C01337=1036.487,-121.338,423.207,168.062,37.819,157.091
C01338=1036.493,-121.088,423.198,168.065,37.818,157.091
C01339=1036.499,-120.839,423.189,168.068,37.817,157.091
C01340=1036.505,-120.588,423.180,168.070,37.816,157.091
C01341=1036.511,-120.338,423.171,168.073,37.815,157.091
C01342=1036.516,-120.089,423.161,168.076,37.814,157.090
C01343=1036.523,-119.839,423.153,168.079,37.813,157.090
C01344=1036.529,-119.589,423.144,168.082,37.812,157.090
C01345=1036.535,-119.340,423.134,168.084,37.811,157.090
C01346=1036.541,-119.090,423.126,168.087,37.810,157.090
C01347=1036.547,-118.840,423.116,168.089,37.809,157.090
C01348=1036.552,-118.590,423.107,168.092,37.808,157.090
C01349=1036.559,-118.341,423.099,168.094,37.808,157.090
C01350=1036.565,-118.091,423.089,168.097,37.806,157.089
C01351=1036.570,-117.841,423.080,168.100,37.805,157.089
C01352=1036.577,-117.592,423.071,168.103,37.805,157.089
C01353=1036.583,-117.342,423.061,168.105,37.804,157.089
C01354=1036.589,-117.092,423.052,168.108,37.802,157.089
C01355=1036.594,-116.842,423.043,168.111,37.802,157.089
C01356=1036.602,-116.556,423.033,168.113,37.801,157.089
C01357=1036.608,-116.269,423.022,168.116,37.799,157.089
C01358=1036.615,-115.983,423.011,168.119,37.799,157.088
C01359=1036.623,-115.696,423.001,168.123,37.798,157.088
C01360=1036.629,-115.447,422.991,168.125,37.796,157.088
C01361=1036.635,-115.197,422.982,168.128,37.796,157.088
C01362=1036.640,-114.947,422.973,168.131,37.795,157.088
C01363=1036.646,-114.697,422.964,168.134,37.794,157.088
C01364=1036.653,-114.448,422.954,168.136,37.793,157.088
C01365=1036.659,-114.198,422.945,168.139,37.792,157.088
C01366=1036.664,-113.949,422.935,168.141,37.791,157.088
C01367=1036.670,-113.698,422.927,168.144,37.791,157.087
C01368=1036.676,-113.448,422.917,168.146,37.790,157.087
C01369=1036.682,-113.199,422.907,168.149,37.789,157.087
C01370=1036.689,-112.949,422.898,168.152,37.788,157.087
C01371=1036.694,-112.700,422.889,168.155,37.787,157.087
C01372=1036.700,-112.450,422.879,168.157,37.786,157.087
C01373=1036.707,-112.200,422.870,168.160,37.785,157.087
C01374=1036.713,-111.950,422.860,168.163,37.785,157.087
C01375=1036.719,-111.701,422.850,168.166,37.784,157.087
C01376=1036.725,-111.450,422.842,168.168,37.783,157.086
C01377=1036.730,-111.201,422.832,168.170,37.782,157.086
C01378=1036.737,-110.951,422.823,168.173,37.782,157.086
C01379=1036.743,-110.701,422.813,168.175,37.781,157.086
C01380=1036.749,-110.452,422.804,168.178,37.780,157.086
C01381=1036.755,-110.202,422.794,168.181,37.779,157.086
C01382=1036.761,-109.952,422.785,168.184,37.778,157.086
C01383=1036.767,-109.702,422.775,168.186,37.777,157.086
C01384=1036.773,-109.453,422.766,168.189,37.776,157.086
C01385=1036.779,-109.203,422.756,168.192,37.776,157.086
C01386=1036.785,-108.953,422.746,168.195,37.775,157.085
C01387=1036.791,-108.703,422.737,168.197,37.774,157.085
C01388=1036.797,-108.454,422.727,168.200,37.773,157.085
C01389=1036.803,-108.204,422.717,168.202,37.773,157.085
C01390=1036.809,-107.954,422.708,168.204,37.772,157.085
C01391=1036.815,-107.704,422.698,168.207,37.771,157.085
C01392=1036.822,-107.454,422.689,168.210,37.770,157.085
C01393=1036.828,-107.205,422.679,168.213,37.770,157.085
C01394=1036.834,-106.955,422.669,168.215,37.769,157.085
C01395=1036.840,-106.705,422.659,168.218,37.768,157.085
C01396=1036.845,-106.456,422.649,168.221,37.767,157.085
C01397=1036.851,-106.206,422.640,168.223,37.767,157.084
C01398=1036.858,-105.957,422.630,168.226,37.766,157.084
C01399=1036.864,-105.707,422.621,168.229,37.765,157.084
C01400=1036.869,-105.457,422.611,168.232,37.764,157.084
C01401=1036.875,-105.207,422.601,168.234,37.764,157.084
C01402=1036.882,-104.958,422.591,168.236,37.763,157.084
C01403=1036.888,-104.708,422.581,168.239,37.762,157.084
C01404=1036.894,-104.458,422.572,168.241,37.761,157.084
C01405=1036.900,-104.208,422.561,168.244,37.761,157.084
C01406=1036.906,-103.958,422.552,168.247,37.761,157.084
C01407=1036.912,-103.709,422.542,168.249,37.760,157.084
C01408=1036.918,-103.459,422.532,168.252,37.759,157.084
C01409=1036.924,-103.209,422.522,168.255,37.758,157.083
C01410=1036.930,-102.959,422.512,168.258,37.758,157.083
C01411=1036.937,-102.710,422.502,168.260,37.757,157.083
C01412=1036.943,-102.460,422.492,168.263,37.756,157.083
C01413=1036.948,-102.210,422.482,168.266,37.755,157.083
C01414=1036.954,-101.961,422.473,168.268,37.755,157.083
C01415=1036.961,-101.711,422.462,168.271,37.754,157.083
C01416=1036.966,-101.461,422.452,168.274,37.754,157.083
C01417=1036.972,-101.211,422.443,168.275,37.753,157.083
C01418=1036.979,-100.962,422.432,168.278,37.752,157.083
C01419=1036.985,-100.712,422.423,168.281,37.751,157.083
C01420=1036.992,-100.425,422.411,168.284,37.751,157.083
C01421=1036.999,-100.137,422.400,168.287,37.750,157.083
C01422=1037.006,-99.850,422.389,168.290,37.749,157.082
C01423=1037.013,-99.563,422.376,168.293,37.748,157.082
C01424=1037.019,-99.313,422.366,168.296,37.748,157.082
C01425=1037.025,-99.064,422.357,168.298,37.747,157.082
C01426=1037.031,-98.814,422.346,168.301,37.747,157.082
C01427=1037.037,-98.564,422.336,168.304,37.746,157.082
C01428=1037.044,-98.315,422.326,168.306,37.745,157.082
C01429=1037.049,-98.065,422.316,168.309,37.745,157.082
C01430=1037.055,-97.815,422.306,168.312,37.744,157.082
C01431=1037.062,-97.566,422.296,168.314,37.743,157.082
C01432=1037.067,-97.316,422.286,168.316,37.743,157.082
C01433=1037.074,-97.066,422.275,168.319,37.742,157.082
C01434=1037.080,-96.816,422.265,168.321,37.742,157.082
C01435=1037.086,-96.567,422.255,168.324,37.741,157.082
C01436=1037.092,-96.317,422.245,168.327,37.741,157.081
C01437=1037.098,-96.067,422.234,168.329,37.740,157.081
C01438=1037.104,-95.817,422.224,168.332,37.740,157.081
C01439=1037.109,-95.568,422.213,168.335,37.739,157.081
C01440=1037.116,-95.318,422.204,168.337,37.739,157.081
C01441=1037.121,-95.069,422.193,168.340,37.738,157.081
C01442=1037.128,-94.818,422.183,168.342,37.738,157.081
C01443=1037.134,-94.569,422.172,168.345,37.737,157.081
C01444=1037.140,-94.319,422.162,168.348,37.737,157.081
C01445=1037.146,-94.069,422.152,168.350,37.736,157.081
C01446=1037.151,-93.820,422.141,168.353,37.736,157.081
C01447=1037.158,-93.570,422.131,168.356,37.735,157.081
C01448=1037.163,-93.321,422.120,168.358,37.734,157.081
C01449=1037.170,-93.071,422.110,168.361,37.734,157.081
C01450=1037.176,-92.821,422.100,168.364,37.734,157.081
C01451=1037.182,-92.571,422.089,168.366,37.734,157.081
C01452=1037.188,-92.322,422.078,168.369,37.733,157.081
C01453=1037.194,-92.072,422.068,168.370,37.732,157.081
C01454=1037.201,-91.822,422.058,168.373,37.732,157.081
C01455=1037.206,-91.572,422.047,168.376,37.731,157.081
C01456=1037.213,-91.323,422.037,168.378,37.731,157.081
C01457=1037.218,-91.073,422.026,168.381,37.730,157.080
C01458=1037.224,-90.824,422.015,168.384,37.730,157.080
C01459=1037.231,-90.574,422.005,168.386,37.730,157.080
C01460=1037.237,-90.324,421.995,168.389,37.729,157.080
C01461=1037.243,-90.074,421.984,168.391,37.729,157.080
C01462=1037.249,-89.825,421.973,168.394,37.728,157.080
C01463=1037.255,-89.574,421.963,168.397,37.727,157.080
C01464=1037.261,-89.325,421.953,168.399,37.727,157.080
C01465=1037.267,-89.075,421.942,168.402,37.726,157.080
C01466=1037.273,-88.826,421.931,168.404,37.726,157.080
C01467=1037.280,-88.576,421.920,168.407,37.726,157.080
C01468=1037.285,-88.326,421.910,168.410,37.725,157.080
C01469=1037.292,-88.077,421.900,168.412,37.725,157.080
C01470=1037.297,-87.827,421.889,168.415,37.724,157.080
C01471=1037.305,-87.577,421.878,168.418,37.724,157.080
C01472=1037.310,-87.328,421.867,168.420,37.723,157.080
C01473=1037.316,-87.078,421.857,168.423,37.723,157.080
C01474=1037.323,-86.828,421.847,168.425,37.722,157.080
C01475=1037.329,-86.578,421.836,168.428,37.722,157.080
C01476=1037.334,-86.329,421.825,168.431,37.722,157.080
C01477=1037.341,-86.079,421.814,168.432,37.721,157.079
C01478=1037.347,-85.830,421.803,168.435,37.721,157.080
C01479=1037.354,-85.580,421.793,168.437,37.720,157.079
C01480=1037.360,-85.330,421.782,168.440,37.720,157.079
C01481=1037.365,-85.080,421.772,168.443,37.719,157.079
C01482=1037.372,-84.831,421.761,168.445,37.719,157.079
C01483=1037.378,-84.581,421.750,168.448,37.718,157.079
C01484=1037.385,-84.296,421.738,168.451,37.718,157.079
C01485=1037.393,-84.011,421.725,168.454,37.717,157.079
C01486=1037.399,-83.727,421.713,168.457,37.717,157.079
C01487=1037.407,-83.441,421.701,168.460,37.717,157.079
C01488=1037.412,-83.192,421.690,168.462,37.716,157.079
C01489=1037.419,-82.942,421.679,168.465,37.716,157.079
C01490=1037.425,-82.693,421.668,168.468,37.715,157.079
C01491=1037.431,-82.442,421.657,168.470,37.715,157.079
C01492=1037.437,-82.193,421.646,168.473,37.714,157.079
C01493=1037.444,-81.944,421.636,168.475,37.714,157.079
C01494=1037.450,-81.693,421.625,168.478,37.713,157.079
C01495=1037.456,-81.444,421.614,168.481,37.713,157.079
C01496=1037.463,-81.194,421.603,168.483,37.713,157.079
C01497=1037.469,-80.945,421.592,168.486,37.712,157.079
C01498=1037.475,-80.694,421.581,168.488,37.712,157.079
C01499=1037.481,-80.445,421.571,168.491,37.711,157.079
C01500=1037.488,-80.195,421.560,168.493,37.711,157.079
C01501=1037.493,-79.946,421.549,168.496,37.710,157.079
C01502=1037.501,-79.696,421.538,168.499,37.710,157.079
C01503=1037.506,-79.446,421.527,168.501,37.710,157.079
C01504=1037.512,-79.197,421.516,168.503,37.709,157.078
C01505=1037.519,-78.947,421.504,168.506,37.709,157.078
C01506=1037.524,-78.698,421.494,168.509,37.709,157.079
C01507=1037.531,-78.447,421.482,168.510,37.708,157.078
C01508=1037.537,-78.198,421.471,168.513,37.708,157.078
C01509=1037.543,-77.948,421.460,168.515,37.708,157.078
C01510=1037.549,-77.699,421.449,168.518,37.708,157.078
C01511=1037.555,-77.449,421.437,168.521,37.707,157.078
C01512=1037.561,-77.199,421.426,168.523,37.707,157.078
C01513=1037.567,-76.949,421.415,168.526,37.707,157.078
C01514=1037.573,-76.700,421.404,168.528,37.707,157.078
C01515=1037.580,-76.450,421.393,168.531,37.706,157.078
C01516=1037.586,-76.201,421.382,168.533,37.706,157.078
C01517=1037.593,-75.951,421.371,168.536,37.706,157.078
C01518=1037.598,-75.701,421.360,168.538,37.706,157.078
C01519=1037.605,-75.452,421.348,168.541,37.706,157.078
C01520=1037.611,-75.202,421.337,168.543,37.705,157.078
C01521=1037.617,-74.952,421.326,168.546,37.705,157.078
C01522=1037.623,-74.703,421.314,168.548,37.705,157.078
C01523=1037.629,-74.453,421.303,168.551,37.704,157.078
C01524=1037.635,-74.203,421.292,168.554,37.704,157.078
C01525=1037.642,-73.954,421.280,168.556,37.704,157.078
C01526=1037.648,-73.704,421.269,168.559,37.704,157.078
C01527=1037.654,-73.454,421.258,168.561,37.704,157.078
C01528=1037.659,-73.205,421.246,168.564,37.703,157.078
C01529=1037.665,-72.955,421.235,168.566,37.703,157.078
C01530=1037.672,-72.705,421.223,168.569,37.703,157.078
C01531=1037.678,-72.456,421.212,168.571,37.703,157.078
C01532=1037.684,-72.205,421.201,168.573,37.703,157.078
C01533=1037.690,-71.956,421.188,168.576,37.702,157.078
C01534=1037.696,-71.706,421.177,168.578,37.702,157.078
C01535=1037.702,-71.457,421.166,168.581,37.702,157.078
C01536=1037.708,-71.207,421.154,168.583,37.702,157.078
C01537=1037.714,-70.958,421.143,168.586,37.701,157.078
C01538=1037.720,-70.708,421.131,168.588,37.701,157.078
C01539=1037.726,-70.459,421.119,168.591,37.701,157.078
C01540=1037.732,-70.209,421.108,168.593,37.701,157.078
C01541=1037.739,-69.959,421.096,168.596,37.701,157.078
C01542=1037.744,-69.709,421.085,168.598,37.701,157.078
C01543=1037.751,-69.460,421.073,168.601,37.701,157.078
C01544=1037.756,-69.210,421.062,168.603,37.701,157.078
C01545=1037.763,-68.961,421.050,168.606,37.701,157.078
C01546=1037.769,-68.710,421.038,168.608,37.701,157.078
C01547=1037.775,-68.461,421.026,168.611,37.701,157.078
C01548=1037.782,-68.178,421.013,168.613,37.701,157.078
C01549=1037.789,-67.895,421.000,168.616,37.700,157.078
C01550=1037.795,-67.612,420.987,168.619,37.700,157.078
C01551=1037.802,-67.330,420.973,168.622,37.700,157.078
C01552=1037.809,-67.080,420.962,168.624,37.700,157.078
C01553=1037.815,-66.831,420.950,168.627,37.700,157.078
C01554=1037.820,-66.581,420.939,168.629,37.699,157.078
C01555=1037.827,-66.331,420.927,168.632,37.699,157.078
C01556=1037.834,-66.082,420.915,168.634,37.699,157.078
C01557=1037.840,-65.832,420.904,168.637,37.699,157.078
C01558=1037.845,-65.582,420.891,168.639,37.699,157.079
C01559=1037.852,-65.333,420.879,168.642,37.699,157.079
C01560=1037.858,-65.083,420.868,168.644,37.699,157.079
C01561=1037.864,-64.833,420.856,168.647,37.699,157.079
C01562=1037.870,-64.584,420.844,168.649,37.699,157.079
C01563=1037.877,-64.334,420.833,168.651,37.699,157.079
C01564=1037.883,-64.085,420.821,168.654,37.698,157.079
C01565=1037.889,-63.835,420.809,168.656,37.698,157.079
C01566=1037.895,-63.585,420.797,168.659,37.698,157.079
C01567=1037.902,-63.335,420.785,168.661,37.698,157.079
C01568=1037.908,-63.086,420.774,168.664,37.698,157.079
C01569=1037.914,-62.836,420.761,168.666,37.698,157.079
C01570=1037.920,-62.587,420.749,168.669,37.698,157.079
C01571=1037.927,-62.337,420.738,168.671,37.698,157.079
C01572=1037.932,-62.087,420.726,168.674,37.697,157.079
C01573=1037.939,-61.838,420.714,168.676,37.697,157.079
C01574=1037.945,-61.588,420.702,168.678,37.697,157.079
C01575=1037.952,-61.338,420.691,168.681,37.697,157.079
C01576=1037.957,-61.089,420.678,168.683,37.697,157.079
C01577=1037.963,-60.839,420.667,168.686,37.697,157.079
C01578=1037.970,-60.590,420.655,168.688,37.697,157.079
C01579=1037.976,-60.340,420.642,168.691,37.697,157.079
C01580=1037.983,-60.090,420.630,168.693,37.697,157.079
C01581=1037.988,-59.841,420.619,168.696,37.697,157.079
C01582=1037.994,-59.591,420.607,168.698,37.697,157.079
C01583=1038.001,-59.341,420.595,168.700,37.697,157.079
C01584=1038.008,-59.092,420.583,168.703,37.697,157.079
C01585=1038.014,-58.842,420.570,168.705,37.696,157.079
C01586=1038.020,-58.592,420.558,168.708,37.696,157.079
C01587=1038.026,-58.343,420.547,168.710,37.696,157.079
C01588=1038.032,-58.094,420.534,168.714,37.696,157.079
C01589=1038.039,-57.844,420.522,168.716,37.696,157.079
C01590=1038.045,-57.594,420.510,168.719,37.696,157.079
C01591=1038.051,-57.344,420.498,168.721,37.696,157.079
C01592=1038.058,-57.094,420.486,168.723,37.696,157.079
C01593=1038.064,-56.845,420.474,168.726,37.696,157.079
C01594=1038.070,-56.595,420.462,168.728,37.696,157.079
C01595=1038.076,-56.346,420.450,168.731,37.696,157.079
C01596=1038.083,-56.096,420.438,168.733,37.696,157.079
C01597=1038.089,-55.847,420.426,168.736,37.696,157.079
C01598=1038.095,-55.597,420.414,168.738,37.695,157.079
C01599=1038.102,-55.347,420.402,168.740,37.695,157.079
C01600=1038.108,-55.098,420.389,168.743,37.695,157.079
C01601=1038.115,-54.848,420.377,168.745,37.695,157.079
C01602=1038.121,-54.598,420.365,168.748,37.695,157.079
C01603=1038.127,-54.348,420.353,168.750,37.695,157.079
C01604=1038.134,-54.099,420.341,168.752,37.695,157.079
C01605=1038.141,-53.849,420.329,168.755,37.695,157.079
C01606=1038.146,-53.599,420.316,168.757,37.695,157.079
C01607=1038.153,-53.351,420.304,168.760,37.695,157.079
C01608=1038.160,-53.101,420.292,168.762,37.695,157.079
C01609=1038.166,-52.851,420.279,168.765,37.695,157.079
C01610=1038.173,-52.601,420.267,168.767,37.695,157.079
C01611=1038.178,-52.352,420.255,168.769,37.695,157.079
C01612=1038.186,-52.071,420.242,168.772,37.694,157.079
C01613=1038.193,-51.789,420.227,168.775,37.694,157.079
C01614=1038.200,-51.507,420.214,168.778,37.694,157.079
C01615=1038.207,-51.226,420.199,168.780,37.694,157.079
C01616=1038.214,-50.976,420.187,168.783,37.694,157.080
C01617=1038.221,-50.727,420.175,168.785,37.694,157.080
C01618=1038.227,-50.477,420.163,168.788,37.694,157.080
C01619=1038.233,-50.227,420.150,168.790,37.694,157.080
C01620=1038.240,-49.978,420.138,168.792,37.694,157.080
C01621=1038.245,-49.728,420.125,168.795,37.694,157.080
C01622=1038.251,-49.478,420.112,168.797,37.694,157.080
C01623=1038.258,-49.228,420.100,168.799,37.694,157.080
C01624=1038.264,-48.979,420.087,168.802,37.694,157.080
C01625=1038.270,-48.729,420.075,168.804,37.695,157.080
C01626=1038.276,-48.479,420.062,168.806,37.695,157.080
C01627=1038.283,-48.230,420.049,168.809,37.695,157.080
C01628=1038.289,-47.981,420.037,168.811,37.695,157.080
C01629=1038.295,-47.731,420.024,168.813,37.695,157.080
C01630=1038.301,-47.481,420.011,168.816,37.695,157.080
C01631=1038.308,-47.232,419.999,168.818,37.695,157.080
C01632=1038.314,-46.982,419.987,168.820,37.695,157.080
C01633=1038.320,-46.733,419.973,168.823,37.695,157.080
C01634=1038.326,-46.483,419.961,168.825,37.695,157.080
C01635=1038.332,-46.233,419.949,168.827,37.695,157.080
C01636=1038.339,-45.984,419.935,168.830,37.695,157.080
C01637=1038.344,-45.734,419.923,168.832,37.696,157.080
C01638=1038.351,-45.485,419.910,168.834,37.696,157.081
C01639=1038.357,-45.235,419.898,168.837,37.696,157.081
C01640=1038.363,-44.985,419.885,168.840,37.696,157.081
C01641=1038.369,-44.736,419.872,168.842,37.696,157.081
C01642=1038.376,-44.487,419.860,168.845,37.696,157.081
C01643=1038.382,-44.237,419.847,168.847,37.696,157.081
C01644=1038.388,-43.987,419.834,168.849,37.697,157.081
C01645=1038.394,-43.738,419.821,168.852,37.697,157.081
C01646=1038.400,-43.488,419.808,168.854,37.696,157.081
C01647=1038.408,-43.239,419.795,168.856,37.696,157.081
C01648=1038.414,-42.989,419.783,168.859,37.697,157.081
C01649=1038.420,-42.739,419.770,168.861,37.697,157.081
C01650=1038.426,-42.490,419.757,168.863,37.697,157.081
C01651=1038.433,-42.240,419.745,168.866,37.697,157.081
C01652=1038.439,-41.991,419.732,168.868,37.697,157.081
C01653=1038.445,-41.742,419.718,168.870,37.697,157.081
C01654=1038.451,-41.492,419.706,168.873,37.697,157.081
C01655=1038.458,-41.242,419.693,168.875,37.698,157.081
C01656=1038.464,-40.992,419.680,168.877,37.698,157.081
C01657=1038.471,-40.743,419.667,168.880,37.698,157.081
C01658=1038.476,-40.493,419.654,168.882,37.698,157.082
C01659=1038.483,-40.244,419.641,168.884,37.698,157.082
C01660=1038.489,-39.994,419.629,168.886,37.698,157.082
C01661=1038.496,-39.744,419.616,168.889,37.698,157.082
C01662=1038.502,-39.495,419.602,168.891,37.699,157.082
C01663=1038.508,-39.245,419.590,168.893,37.698,157.082
C01664=1038.514,-38.996,419.576,168.896,37.698,157.082
C01665=1038.521,-38.746,419.564,168.898,37.699,157.082
C01666=1038.528,-38.496,419.551,168.900,37.699,157.082
C01667=1038.533,-38.247,419.537,168.904,37.699,157.082
C01668=1038.539,-37.997,419.524,168.906,37.699,157.082
C01669=1038.546,-37.747,419.511,168.908,37.699,157.082
C01670=1038.552,-37.498,419.498,168.910,37.700,157.082
C01671=1038.559,-37.248,419.484,168.913,37.700,157.082
C01672=1038.564,-36.998,419.472,168.915,37.700,157.082
C01673=1038.571,-36.749,419.458,168.917,37.700,157.082
C01674=1038.577,-36.500,419.445,168.919,37.701,157.083
C01675=1038.583,-36.250,419.433,168.922,37.701,157.083
C01676=1038.590,-35.969,419.417,168.924,37.701,157.083
C01677=1038.597,-35.687,419.402,168.927,37.701,157.083
C01678=1038.604,-35.407,419.388,168.929,37.702,157.083
C01679=1038.612,-35.126,419.373,168.932,37.702,157.083
C01680=1038.618,-34.877,419.360,168.934,37.702,157.083
C01681=1038.625,-34.627,419.346,168.936,37.702,157.083
C01682=1038.631,-34.377,419.333,168.939,37.703,157.083
C01683=1038.636,-34.127,419.320,168.941,37.703,157.083
C01684=1038.642,-33.878,419.307,168.943,37.703,157.083
C01685=1038.649,-33.628,419.293,168.945,37.703,157.083
C01686=1038.655,-33.379,419.280,168.949,37.703,157.083
C01687=1038.661,-33.129,419.266,168.951,37.704,157.083
C01688=1038.668,-32.879,419.253,168.953,37.704,157.084
C01689=1038.674,-32.630,419.240,168.955,37.704,157.084
C01690=1038.680,-32.380,419.227,168.958,37.704,157.084
C01691=1038.687,-32.131,419.214,168.960,37.705,157.084
C01692=1038.693,-31.881,419.200,168.962,37.705,157.084
C01693=1038.700,-31.632,419.187,168.964,37.705,157.084
C01694=1038.706,-31.383,419.174,168.967,37.705,157.084
C01695=1038.713,-31.133,419.160,168.969,37.706,157.084
C01696=1038.719,-30.883,419.147,168.971,37.706,157.084
C01697=1038.725,-30.634,419.133,168.973,37.706,157.084
C01698=1038.731,-30.384,419.119,168.976,37.706,157.084
C01699=1038.737,-30.135,419.106,168.978,37.706,157.084
C01700=1038.743,-29.885,419.093,168.980,37.707,157.084
C01701=1038.750,-29.635,419.080,168.982,37.707,157.084
C01702=1038.756,-29.385,419.066,168.985,37.707,157.085
C01703=1038.762,-29.136,419.053,168.987,37.707,157.085
C01704=1038.769,-28.886,419.040,168.990,37.708,157.085
C01705=1038.775,-28.637,419.026,168.992,37.708,157.085
C01706=1038.782,-28.388,419.013,168.994,37.708,157.085
C01707=1038.789,-28.138,418.999,168.997,37.708,157.085
C01708=1038.795,-27.888,418.986,168.999,37.709,157.085
C01709=1038.801,-27.638,418.972,169.001,37.709,157.085
C01710=1038.807,-27.389,418.959,169.003,37.709,157.085
C01711=1038.813,-27.140,418.945,169.006,37.709,157.085
C01712=1038.820,-26.890,418.931,169.008,37.709,157.085
C01713=1038.827,-26.641,418.918,169.010,37.710,157.085
C01714=1038.833,-26.391,418.903,169.012,37.710,157.085
C01715=1038.839,-26.142,418.890,169.014,37.710,157.086
C01716=1038.845,-25.892,418.877,169.017,37.711,157.086
C01717=1038.851,-25.642,418.863,169.019,37.711,157.086
C01718=1038.857,-25.393,418.849,169.021,37.711,157.086
C01719=1038.864,-25.143,418.836,169.023,37.712,157.086
C01720=1038.870,-24.894,418.821,169.025,37.712,157.086
C01721=1038.876,-24.645,418.808,169.028,37.712,157.086
C01722=1038.883,-24.395,418.794,169.031,37.713,157.086
C01723=1038.888,-24.145,418.780,169.033,37.713,157.086
C01724=1038.895,-23.895,418.767,169.035,37.714,157.086
C01725=1038.901,-23.645,418.753,169.037,37.714,157.087
C01726=1038.907,-23.397,418.739,169.039,37.714,157.087
C01727=1038.914,-23.147,418.725,169.042,37.715,157.087
C01728=1038.920,-22.897,418.711,169.044,37.715,157.087
C01729=1038.926,-22.647,418.698,169.046,37.715,157.087
C01730=1038.933,-22.399,418.684,169.048,37.716,157.087
C01731=1038.939,-22.148,418.670,169.050,37.716,157.087
C01732=1038.945,-21.899,418.656,169.052,37.716,157.087
C01733=1038.951,-21.650,418.643,169.055,37.717,157.087
C01734=1038.958,-21.400,418.628,169.057,37.717,157.087
C01735=1038.964,-21.151,418.615,169.059,37.717,157.087
C01736=1038.970,-20.901,418.601,169.061,37.717,157.087
C01737=1038.977,-20.652,418.587,169.064,37.718,157.088
C01738=1038.983,-20.402,418.573,169.066,37.718,157.088
C01739=1038.989,-20.152,418.559,169.069,37.718,157.088
C01740=1038.996,-19.871,418.543,169.071,37.719,157.088
C01741=1039.004,-19.588,418.528,169.074,37.720,157.088
C01742=1039.011,-19.307,418.512,169.076,37.719,157.088
C01743=1039.018,-19.025,418.496,169.078,37.720,157.088
C01744=1039.025,-18.775,418.482,169.081,37.721,157.088
C01745=1039.030,-18.526,418.468,169.083,37.721,157.088
C01746=1039.038,-18.276,418.454,169.085,37.721,157.088
C01747=1039.044,-18.027,418.441,169.087,37.722,157.089
C01748=1039.050,-17.777,418.426,169.089,37.722,157.089
C01749=1039.056,-17.528,418.412,169.091,37.722,157.089
C01750=1039.062,-17.278,418.398,169.094,37.723,157.089
C01751=1039.069,-17.029,418.384,169.097,37.723,157.089
C01752=1039.076,-16.779,418.371,169.099,37.723,157.089
C01753=1039.082,-16.529,418.356,169.101,37.723,157.089
C01754=1039.088,-16.280,418.342,169.103,37.724,157.089
C01755=1039.094,-16.030,418.328,169.105,37.724,157.089
C01756=1039.101,-15.781,418.314,169.107,37.724,157.089
C01757=1039.107,-15.531,418.300,169.110,37.725,157.089
C01758=1039.114,-15.283,418.286,169.112,37.725,157.090
C01759=1039.120,-15.032,418.272,169.114,37.725,157.090
C01760=1039.127,-14.783,418.257,169.116,37.726,157.090
C01761=1039.132,-14.533,418.243,169.118,37.727,157.090
C01762=1039.139,-14.284,418.229,169.120,37.727,157.090
C01763=1039.145,-14.034,418.215,169.122,37.727,157.090
C01764=1039.151,-13.785,418.200,169.124,37.728,157.090
C01765=1039.158,-13.536,418.186,169.127,37.728,157.090
C01766=1039.164,-13.286,418.172,169.130,37.729,157.090
C01767=1039.170,-13.036,418.157,169.132,37.729,157.091
C01768=1039.176,-12.787,418.144,169.134,37.729,157.091
C01769=1039.183,-12.537,418.129,169.136,37.730,157.091
C01770=1039.188,-12.288,418.115,169.138,37.730,157.091
C01771=1039.195,-12.038,418.101,169.140,37.731,157.091
C01772=1039.202,-11.789,418.086,169.142,37.731,157.091
C01773=1039.207,-11.539,418.072,169.144,37.732,157.091
C01774=1039.214,-11.290,418.058,169.146,37.732,157.091
C01775=1039.220,-11.041,418.043,169.148,37.733,157.091
C01776=1039.226,-10.791,418.029,169.151,37.733,157.091
C01777=1039.233,-10.541,418.014,169.154,37.733,157.092
C01778=1039.239,-10.292,418.000,169.156,37.734,157.092
C01779=1039.245,-10.042,417.986,169.158,37.734,157.092
C01780=1039.252,-9.793,417.971,169.160,37.735,157.092
C01781=1039.258,-9.544,417.957,169.162,37.735,157.092
C01782=1039.264,-9.293,417.942,169.164,37.735,157.092
C01783=1039.271,-9.044,417.928,169.166,37.736,157.092
C01784=1039.277,-8.795,417.914,169.168,37.737,157.092
C01785=1039.283,-8.545,417.899,169.170,37.737,157.092
C01786=1039.290,-8.295,417.885,169.172,37.737,157.092
C01787=1039.296,-8.047,417.870,169.175,37.738,157.093
C01788=1039.302,-7.797,417.855,169.177,37.738,157.093
C01789=1039.309,-7.547,417.840,169.179,37.738,157.093
C01790=1039.316,-7.297,417.827,169.182,37.739,157.093
C01791=1039.321,-7.048,417.812,169.184,37.739,157.093
C01792=1039.328,-6.799,417.797,169.186,37.740,157.093
C01793=1039.335,-6.549,417.783,169.188,37.740,157.093
C01794=1039.340,-6.300,417.769,169.190,37.740,157.093
C01795=1039.347,-6.050,417.754,169.192,37.741,157.093
C01796=1039.354,-5.801,417.740,169.194,37.742,157.094
C01797=1039.360,-5.551,417.725,169.196,37.742,157.094
C01798=1039.366,-5.302,417.710,169.198,37.742,157.094
C01799=1039.373,-5.053,417.696,169.201,37.743,157.094
C01800=1039.379,-4.802,417.682,169.203,37.743,157.094
C01801=1039.386,-4.553,417.667,169.206,37.744,157.094
C01802=1039.391,-4.304,417.652,169.208,37.744,157.094
C01803=1039.399,-4.054,417.638,169.210,37.744,157.094
C01804=1039.406,-3.771,417.621,169.212,37.745,157.094
C01805=1039.413,-3.487,417.605,169.215,37.745,157.095
C01806=1039.420,-3.204,417.587,169.217,37.746,157.095
C01807=1039.427,-2.920,417.571,169.219,37.747,157.095
C01808=1039.433,-2.671,417.556,169.221,37.747,157.095
C01809=1039.439,-2.422,417.541,169.223,37.748,157.095
C01810=1039.446,-2.172,417.526,169.225,37.748,157.095
C01811=1039.452,-1.922,417.511,169.227,37.749,157.095
C01812=1039.458,-1.673,417.496,169.230,37.750,157.096
C01813=1039.464,-1.424,417.482,169.232,37.750,157.096
C01814=1039.471,-1.174,417.467,169.234,37.751,157.096
